# B&R Automation Studio project NAEUL004C00R13L518F00 (part 24)

#### Act_OptP1020Navi.st
```iecst
ACTION Act_OptP1020Navi:

	IF tyP1020McSetNavi.tyNavi.tyBtnMcSet.bRtCompl = TRUE THEN
		tyP1020McSetNavi.tyNavi.tyBtnMcSet.bRtCompl			:= FALSE;
		tyP1020McSetNavi.tyNavi.tyBtnMcSet.bValue			:= FALSE;

		eChgPage	:= UIP1021McSetGen;

	ELSIF tyP1020McSetNavi.tyNavi.tyBtnVCommSet.bRtCompl = TRUE THEN
		tyP1020McSetNavi.tyNavi.tyBtnVCommSet.bRtCompl		:= FALSE;
		tyP1020McSetNavi.tyNavi.tyBtnVCommSet.bValue		:= FALSE;

		eChgPage	:= UIP1022McSetVComm;

	ELSIF tyP1020McSetNavi.tyNavi.tyBtnHCommSet.bRtCompl = TRUE THEN
		tyP1020McSetNavi.tyNavi.tyBtnHCommSet.bRtCompl		:= FALSE;
		tyP1020McSetNavi.tyNavi.tyBtnHCommSet.bValue		:= FALSE;

		eChgPage	:= UIP1023McSetHComm;

	ELSIF tyP1020McSetNavi.tyNavi.tyBtnAntiGapSet.bRtCompl = TRUE THEN
		tyP1020McSetNavi.tyNavi.tyBtnAntiGapSet.bRtCompl	:= FALSE;
		tyP1020McSetNavi.tyNavi.tyBtnAntiGapSet.bValue		:= FALSE;

		eChgPage	:= UIP1024McSetAntiGap;

	ELSIF tyP1020McSetNavi.tyNavi.tyBtnScanSet.bRtCompl = TRUE THEN
		tyP1020McSetNavi.tyNavi.tyBtnScanSet.bRtCompl	:= FALSE;
		tyP1020McSetNavi.tyNavi.tyBtnScanSet.bValue		:= FALSE;

		eChgPage	:= UIP1025McSetScan;

	ELSIF tyP1020McSetNavi.tyNavi.tyBtnOpConSet.bRtCompl = TRUE THEN
		tyP1020McSetNavi.tyNavi.tyBtnOpConSet.bRtCompl	:= FALSE;
		tyP1020McSetNavi.tyNavi.tyBtnOpConSet.bValue		:= FALSE;

		eChgPage	:= UIP1027McSetOpCon;
	END_IF

END_ACTION
```

#### Act_EntP1021Disp.st
```iecst
ACTION Act_EntP1021Disp:

	//Access Address
	IF bTeachTravPosA OR bTeachTravPosB OR bTeachLifterPosA OR bTeachLifterPosB THEN
		p_tyC0004Navi ACCESS ADR(tyP1021McSetGen.tyNaviLyr2);
	ELSIF ((p_tyNtParamCurr.bProjMagConvLane1Prep AND p_tyNtParamCurr.bProjMagConvLane2Prep)
		OR bTeachLifterTopPos OR bTeachLifterTopPos2 OR bTeachLifterBtmPos OR bTeachLifterBtmPos2) OR (p_tyNtParamCurr.tyDISettings.diMagWidthChkSen <>0) THEN
		p_tyC0004Navi ACCESS ADR(tyP1021McSetGen.tyNaviLyr3);
	ELSE
		p_tyC0004Navi ACCESS ADR(tyP1021McSetGen.tyNaviLyr1);
	END_IF

	p_tyC0005Main ACCESS ADR(tyCommon.tyMain);

	p_tyC0006Set ACCESS ADR(tyCommon.tySet);

	p_tyC0007Notif ACCESS ADR(tyCommon.tyNotif);

	p_tyC0008MsgBox ACCESS ADR(tyP1021McSetGen.tyMsgBoxHide);

	p_tyC0009Info ACCESS ADR(tyCommon.tyInfo);

	p_tyP1021McSetGen ACCESS ADR(tyP1021McSetGen.tyGen);
	p_tyP1021McSetNetwork ACCESS ADR(tyP1021McSetGen.tyNetwork);

	//Display
//	tyP1021McSetGen.tyGen.tyLyrGen1.uiRtStat.0	:= bTeachTravPosA OR bTeachTravPosB OR bTeachLifterPosA OR bTeachLifterPosB;
//	tyP1021McSetGen.tyGen.tyLyrGen2.uiRtStat.0	:= NOT(bTeachTravPosA OR bTeachTravPosB OR bTeachLifterPosA OR bTeachLifterPosB);

	//Backup Param
	IF NOT(bTeachTravPosA OR bTeachTravPosB OR bTeachLifterPosA OR bTeachLifterPosB OR
		bTeachLifterTopPos OR bTeachLifterBtmPos OR bTeachLifterTopPos2 OR bTeachLifterBtmPos2) THEN
		tyP1021McSetGen.tyGenBkUp	:= tyP1021McSetGen.tyGen;
	ELSE
		bTeachTravPosA		:= FALSE;
		bTeachTravPosB		:= FALSE;
		bTeachLifterPosA	:= FALSE;
		bTeachLifterPosB	:= FALSE;
		bTeachLifterTopPos	:= FALSE;
		bTeachLifterBtmPos	:= FALSE;
		bTeachLifterTopPos2	:= FALSE;
		bTeachLifterBtmPos2	:= FALSE;
	END_IF
	//Network Configuration Display
	usiNetworkModeOld := DINT_TO_USINT(p_tyMcParamCurr.eNetworkMod);

	fUIInRtStatHide(ADR(tyP1021McSetGen.tyNetwork.tyLyr.uiRtStat));

	IF p_tyDI.bInShutterCloseRS THEN
		tyP1021McSetGen.tyGen.tyBtnInShutterDis.uiMaskRtStat.0 := FALSE;
	ELSE
		tyP1021McSetGen.tyGen.tyBtnInShutterDis.uiMaskRtStat.0 := TRUE;
	END_IF

//	//Penumatic
//	tyP1021McSetGen.tyGen.tyBtnInShutterDis.uiRtStat.0 := TRUE;
	tyP1021McSetGen.tyGen.tyBtnStopperADis.uiRtStat.0 := TRUE;
	tyP1021McSetGen.tyGen.tyBtnStopperBDis.uiRtStat.0 := TRUE;

//	CASE p_tyNtParamCurr.eProjMag OF
//		ULMagDual:
//			tyP1021McSetGen.tyGen.tyStringMcNm.sValue := 'Dual Magazine Line Unloader';
//
//		ULMagTriple:
//			tyP1021McSetGen.tyGen.tyStringMcNm.sValue := 'Triple Magazine Line Unloader';
//
//		ULMagQuadruple:
//			tyP1021McSetGen.tyGen.tyStringMcNm.sValue := 'Quadruple Magazine Line Unloader';
//	END_CASE

	tyP1021McSetGen.tyGen.tyBtnLFBuzMute.uiRtStat.0 := NOT (p_tyMcParamCurr.bLFEn AND p_tyNtParamCurr.bLFPrep AND p_tyNtParamCurr.tyDOSettings.diBuzzer > 0);

	//Siemen Request Hide inlet shutter
	IF p_eNtParamCustomerReq = Siemens THEN
		IF p_tyUsrMgmtCurrAccessRgt.bUsrMgmt THEN
			tyP1021McSetGen.tyGen.tyBtnInShutterDis.uiMaskRtStat := TRUE;
		ELSE
			tyP1021McSetGen.tyGen.tyBtnInShutterDis.uiMaskRtStat := FALSE;
		END_IF
	ELSE
		tyP1021McSetGen.tyGen.tyBtnInShutterDis.uiMaskRtStat := TRUE;
	END_IF
	//Siemen update change for RFID
	tyP1021McSetGen.tyGen.tyBtnMESEn.bValue					:= p_tyMcParamCurr.bMESEn;	//RFID
	tyP1021McSetGen.tyGen.tyBtnHermesSvyEn.bValue					:= p_tyMcParamCurr.bHermesSvyEn;	//RFID

END_ACTION
```

#### Act_ExitP1021.st
```iecst
ACTION Act_ExitP1021:

	IF (tyCommon.tySet.tyBtnSave.uiMaskRtStat.0 = FALSE) OR (bTeachTravPosA OR bTeachTravPosB OR bTeachLifterPosA OR bTeachLifterPosB) THEN
		usiChgPage	:= 1;

	ELSE

		p_tyC0008MsgBox ACCESS ADR(tyP1021McSetGen.tyMsgBoxExitAsk);

		IF tyP1021McSetGen.tyMsgBoxExitAsk.tyBtnYes.bRtCompl = TRUE THEN
			tyP1021McSetGen.tyMsgBoxExitAsk.tyBtnYes.bRtCompl	:= FALSE;
			tyP1021McSetGen.tyMsgBoxExitAsk.tyBtnYes.bValue		:= FALSE;

			p_tyC0008MsgBox ACCESS ADR(tyP1021McSetGen.tyMsgBoxHide);

			//Restore Param
			tyP1021McSetGen.tyGen	:= tyP1021McSetGen.tyGenBkUp;

			fUIInRtStatOff(ADR(tyCommon.tySet.tyBtnSave.uiMaskRtStat));

			bSaveNetworkPriority := FALSE;

			usiChgPage	:= 1;

		ELSIF tyP1021McSetGen.tyMsgBoxExitAsk.tyBtnNo.bRtCompl = TRUE THEN
			tyP1021McSetGen.tyMsgBoxExitAsk.tyBtnNo.bRtCompl	:= FALSE;
			tyP1021McSetGen.tyMsgBoxExitAsk.tyBtnNo.bValue		:= FALSE;

			p_tyC0008MsgBox ACCESS ADR(tyP1021McSetGen.tyMsgBoxHide);

			eChgPage	:= eCurrPage;
			usiChgPage	:= 0;

		END_IF

	END_IF

END_ACTION
```

#### Act_OptP1021Navi.st
```iecst
ACTION Act_OptP1021Navi:

	tyP1021McSetGen.tyNaviLyr1.tyBtnBack.bRtLk	:= tyCommon.tySet.tyBtnSave.bRtCompl;
	tyP1021McSetGen.tyNaviLyr2.tyBtnBack.bRtLk	:= tyCommon.tySet.tyBtnSave.bRtCompl;
	tyP1021McSetGen.tyNaviLyr3.tyBtnBack.bRtLk	:= tyCommon.tySet.tyBtnSave.bRtCompl;

	IF tyP1021McSetGen.tyNaviLyr1.tyBtnBack.bRtCompl = TRUE OR tyP1021McSetGen.tyNaviLyr2.tyBtnBack.bRtCompl = TRUE
		OR tyP1021McSetGen.tyNaviLyr3.tyBtnBack.bRtCompl = TRUE THEN
		tyP1021McSetGen.tyNaviLyr1.tyBtnBack.bRtCompl		:= FALSE;
		tyP1021McSetGen.tyNaviLyr2.tyBtnBack.bRtCompl		:= FALSE;
		tyP1021McSetGen.tyNaviLyr3.tyBtnBack.bRtCompl		:= FALSE;

		eChgPage	:= UIP1020McSetNavi;
	END_IF

	IF (p_tyNtParamCurr.bProjMagConvLane1Prep AND p_tyNtParamCurr.bProjMagConvLane2Prep) OR
		(p_tyNtParamCurr.tyDISettings.diMagWidthChkSen <> 0 OR p_tyNtParamCurr.bProjInletStopperPrep
		OR p_tyNtParamCurr.eCustomerReq = Siemens OR p_tyNtParamCurr.bAutoRcpPrep OR p_tyNtParamCurr.tyDISettings.diScanComplSig <> 0)

		THEN
		p_tyC0004Navi ACCESS ADR (tyP1021McSetGen.tyNaviLyr3);
		IF tyP1021McSetGen.tyNaviLyr3.tyBtnRgt.bRtCompl AND tyP1021McSetGen.tyNaviLyr3.tyBitmapPageDisp.usiValueIdx =3
			OR tyP1021McSetGen.tyNaviLyr3.tyBtnLeft.bRtCompl AND tyP1021McSetGen.tyNaviLyr3.tyBitmapPageDisp.usiValueIdx =5 THEN

			tyP1021McSetGen.tyNaviLyr3.tyBitmapPageDisp.usiValueIdx := 4;
			fUIInRtStatHide(ADR(tyP1021McSetGen.tyGen.tyLyrGen1.uiRtStat));
			fUIInRtStatOff(ADR(tyP1021McSetGen.tyGen.tyLyrGen2.uiRtStat));
			fUIInRtStatHide(ADR(tyP1021McSetGen.tyGen.tyLyrGen3.uiRtStat));
			fUIInRtStatHide(ADR(tyP1021McSetGen.tyGen.tyLyrGen4.uiRtStat));
			tyP1021McSetGen.tyNaviLyr3.tyBtnRgt.bRtCompl := FALSE;
			tyP1021McSetGen.tyNaviLyr3.tyBtnLeft.bRtCompl := FALSE;

		ELSIF tyP1021McSetGen.tyNaviLyr3.tyBtnLeft.bRtCompl AND tyP1021McSetGen.tyNaviLyr3.tyBitmapPageDisp.usiValueIdx =3
			OR tyP1021McSetGen.tyNaviLyr3.tyBtnRgt.bRtCompl AND tyP1021McSetGen.tyNaviLyr3.tyBitmapPageDisp.usiValueIdx =4 THEN

			tyP1021McSetGen.tyNaviLyr3.tyBitmapPageDisp.usiValueIdx := 5;
			fUIInRtStatHide(ADR(tyP1021McSetGen.tyGen.tyLyrGen1.uiRtStat));
			fUIInRtStatHide(ADR(tyP1021McSetGen.tyGen.tyLyrGen2.uiRtStat));
			IF (NOT p_tyNtParamCurr.bProjMagConvLane1Prep AND NOT p_tyNtParamCurr.bProjMagConvLane2Prep)
				AND (p_tyNtParamCurr.tyDISettings.diMagWidthChkSen <> 0 OR p_tyNtParamCurr.bProjInletStopperPrep OR p_tyNtParamCurr.eCustomerReq = Siemens OR  p_tyNtParamCurr.eCustomerReq = We_Fabricate ) THEN
				fUIInRtStatHide(ADR(tyP1021McSetGen.tyGen.tyLyrGen3.uiRtStat));
				fUIInRtStatOff(ADR(tyP1021McSetGen.tyGen.tyLyrGen4.uiRtStat));
			ELSE
				fUIInRtStatOff(ADR(tyP1021McSetGen.tyGen.tyLyrGen3.uiRtStat));
				fUIInRtStatHide(ADR(tyP1021McSetGen.tyGen.tyLyrGen4.uiRtStat));
			END_IF

			tyP1021McSetGen.tyNaviLyr3.tyBtnRgt.bRtCompl := FALSE;
			tyP1021McSetGen.tyNaviLyr3.tyBtnLeft.bRtCompl := FALSE;

		ELSIF (tyP1021McSetGen.tyNaviLyr3.tyBtnLeft.bRtCompl AND tyP1021McSetGen.tyNaviLyr3.tyBitmapPageDisp.usiValueIdx =4)
			OR (tyP1021McSetGen.tyNaviLyr3.tyBtnRgt.bRtCompl AND tyP1021McSetGen.tyNaviLyr3.tyBitmapPageDisp.usiValueIdx =5) THEN

			tyP1021McSetGen.tyNaviLyr3.tyBitmapPageDisp.usiValueIdx := 3;
			fUIInRtStatOff(ADR(tyP1021McSetGen.tyGen.tyLyrGen1.uiRtStat));
			fUIInRtStatHide(ADR(tyP1021McSetGen.tyGen.tyLyrGen2.uiRtStat));
			fUIInRtStatHide(ADR(tyP1021McSetGen.tyGen.tyLyrGen3.uiRtStat));
			fUIInRtStatHide(ADR(tyP1021McSetGen.tyGen.tyLyrGen4.uiRtStat));
			tyP1021McSetGen.tyNaviLyr3.tyBtnRgt.bRtCompl := FALSE;
			tyP1021McSetGen.tyNaviLyr3.tyBtnLeft.bRtCompl := FALSE;
		END_IF

	ELSE

		//Navi From Layer 1 to Layer 2
		IF tyP1021McSetGen.tyNaviLyr1.tyBtnRgt.bRtCompl = TRUE THEN
			p_tyC0004Navi ACCESS ADR (tyP1021McSetGen.tyNaviLyr2);

			fUIInRtStatHide(ADR(tyP1021McSetGen.tyGen.tyLyrGen1.uiRtStat));
			fUIInRtStatOff(ADR(tyP1021McSetGen.tyGen.tyLyrGen2.uiRtStat));

			tyP1021McSetGen.tyNaviLyr1.tyBtnRgt.bRtCompl			:= FALSE;

		ELSIF tyP1021McSetGen.tyNaviLyr1.tyBtnLeft.bRtCompl = TRUE THEN
			p_tyC0004Navi ACCESS ADR (tyP1021McSetGen.tyNaviLyr2);

			fUIInRtStatHide(ADR(tyP1021McSetGen.tyGen.tyLyrGen1.uiRtStat));
			fUIInRtStatOff(ADR(tyP1021McSetGen.tyGen.tyLyrGen2.uiRtStat));

			tyP1021McSetGen.tyNaviLyr1.tyBtnLeft.bRtCompl			:= FALSE;

		//Navi Form Layer 2 to Layer 1
		ELSIF tyP1021McSetGen.tyNaviLyr2.tyBtnRgt.bRtCompl = TRUE THEN
			p_tyC0004Navi ACCESS ADR(tyP1021McSetGen.tyNaviLyr1);

			fUIInRtStatOff(ADR(tyP1021McSetGen.tyGen.tyLyrGen1.uiRtStat));
			fUIInRtStatHide(ADR(tyP1021McSetGen.tyGen.tyLyrGen2.uiRtStat));

			tyP1021McSetGen.tyNaviLyr2.tyBtnRgt.bRtCompl			:= FALSE;

		ELSIF tyP1021McSetGen.tyNaviLyr2.tyBtnLeft.bRtCompl = TRUE THEN
			p_tyC0004Navi ACCESS ADR(tyP1021McSetGen.tyNaviLyr1);

			fUIInRtStatOff(ADR(tyP1021McSetGen.tyGen.tyLyrGen1.uiRtStat));
			fUIInRtStatHide(ADR(tyP1021McSetGen.tyGen.tyLyrGen2.uiRtStat));

			tyP1021McSetGen.tyNaviLyr2.tyBtnLeft.bRtCompl			:= FALSE;

		END_IF
	END_IF

END_ACTION
```

#### Act_OptP1021Save.st
```iecst
ACTION Act_OptP1021Save:
		//Only Applicable when next page appears.

	IF p_tyP1021McSetGen.tyDrpDnPos1.uiRtStat.0 = FALSE
		AND p_tyP1021McSetGen.tyDrpDnPos2.uiRtStat.0 = FALSE
		AND p_tyP1021McSetGen.tyDrpDnPos3.uiRtStat.0 = FALSE THEN

		usiDuplicate := 6;

	ELSIF p_tyP1021McSetGen.tyDrpDnPos1.uiRtStat.0 = FALSE
		AND p_tyP1021McSetGen.tyDrpDnPos2.uiRtStat.0 = FALSE
		AND p_tyP1021McSetGen.tyDrpDnPos3.uiRtStat.0 = TRUE THEN

		usiDuplicate := 3;
	END_IF

	IF tyP1021McSetGen.tyGen.tyStringMcNm.bRtCompl
		OR tyP1021McSetGen.tyGen.tyDrpDnDefaultMcMod.bRtCompl	OR tyP1021McSetGen.tyGen.tyNumSSaverTm.bRtCompl
		OR tyP1021McSetGen.tyGen.tyBtnSSaverEn.bRtCompl			OR tyP1021McSetGen.tyGen.tyNumWidthAtHm.bRtCompl
		OR tyP1021McSetGen.tyGen.tyNumConvInitTm.bRtCompl		OR tyP1021McSetGen.tyGen.tyNumTranInErrDlyTm.bRtCompl
		OR tyP1021McSetGen.tyGen.tyNumMag1ConvRunTm.bRtCompl	OR tyP1021McSetGen.tyGen.tyNumMag2ConvRunTm.bRtCompl
		OR tyP1021McSetGen.tyGen.tyNumMag3ConvRunTm.bRtCompl 	OR tyP1021McSetGen.tyGen.tyNumMaxBffr.bRtCompl
		OR tyP1021McSetGen.tyGen.tyNumTravPosLaneA.bRtCompl		OR tyP1021McSetGen.tyGen.tyNumLiftPosLaneA.bRtCompl
		OR tyP1021McSetGen.tyGen.tyNumTravPosLaneB.bRtCompl		OR tyP1021McSetGen.tyGen.tyNumLiftPosLaneB.bRtCompl
		OR tyP1021McSetGen.tyGen.tyBtnAWDis.bRtCompl			OR tyP1021McSetGen.tyGen.tyBtnMnlAccDat.bRtCompl
		OR tyP1021McSetGen.tyGen.tyBtnAutoStepEn.bRtCompl		OR tyP1021McSetGen.tyGen.tyBtnVSMEMAEn.bRtCompl
		OR tyP1021McSetGen.tyGen.tyBtnHermesRmtEn.bRtCompl		OR tyP1021McSetGen.tyGen.tyBtnGapBetBrdEn.bRtCompl
		OR tyP1021McSetGen.tyGen.tyBtnLongBrdEn.bRtCompl		OR tyP1021McSetGen.tyGen.tyBtnOvenEn.bRtCompl
		OR tyP1021McSetGen.tyGen.tyBtnExtdOvenEn.bRtCompl		OR tyP1021McSetGen.tyGen.tyBtnInShutterDis.bRtCompl
		OR tyP1021McSetGen.tyGen.tyBtnChgParamEn.bRtCompl		OR tyP1021McSetGen.tyGen.tyBtnStopperADis.bRtCompl
		OR tyP1021McSetGen.tyGen.tyBtnStopperBDis.bRtCompl 		OR tyP1021McSetGen.tyGen.tyNumWidthOffset.bRtCompl
		OR tyP1021McSetGen.tyGen.tyBtnAGVComEn.bRtCompl  		OR tyP1021McSetGen.tyGen.tyNumMagAutoDetSenTm.bRtCompl
		OR tyP1021McSetGen.tyGen.tyNumMag1WidthAtHm.bRtCompl	OR tyP1021McSetGen.tyGen.tyNumMag2WidthAtHm.bRtCompl
		OR tyP1021McSetGen.tyGen.tyNumMag3WidthAtHm.bRtCompl	OR tyP1021McSetGen.tyGen.tyBtnMagAWDis.bRtCompl
		OR tyP1021McSetGen.tyGen.tyBtnMagSafetyBarDis.bRtCompl 	OR tyP1021McSetGen.tyGen.tyBtnAutoLogoutEn.bRtCompl
		OR tyP1021McSetGen.tyGen.tyNumAutoLogoutTm.bRtCompl		OR tyP1021McSetGen.tyGen.tyBtnLFBuzMute.bRtCompl
		OR tyP1021McSetGen.tyGen.tyDrpDnAGVComProtocol.bRtCompl OR tyP1021McSetGen.tyGen.tyDrpDnMagExchangeMode.bRtCompl
		OR tyP1021McSetGen.tyGen.tyBtnAGVSizeDisabled.bRtCompl
		OR tyP1021McSetGen.tyGen.tyNumAWPusherAtHm.bRtCompl		OR tyP1021McSetGen.tyGen.tyBtnAWPusherDis.bRtCompl
		OR tyP1021McSetGen.tyGen.tyNumTravFixtoFixPosInlet.bRtCompl
		OR tyP1021McSetGen.tyGen.tyBtnDisableFMWarning.bRtCompl
		OR tyP1021McSetGen.tyGen.tyNumInMagConvInitTm.bRtCompl OR tyP1021McSetGen.tyGen.tyNumOutMagConvInitTm.bRtCompl
		OR tyP1021McSetGen.tyGen.tyNumLifterTopPos.bRtCompl OR tyP1021McSetGen.tyGen.tyNumLifterBtmPos.bRtCompl
		OR tyP1021McSetGen.tyGen.tyNumLifterMagConvInitTm.bRtCompl
		OR tyP1021McSetGen.tyGen.tyNumInMagConv2InitTm.bRtCompl OR tyP1021McSetGen.tyGen.tyNumOutMagConv2InitTm.bRtCompl
		OR tyP1021McSetGen.tyGen.tyNumLifterTopPos2.bRtCompl OR tyP1021McSetGen.tyGen.tyNumLifterBtmPos2.bRtCompl
		OR tyP1021McSetGen.tyGen.tyNumLifterMagConv2InitTm.bRtCompl OR tyP1021McSetGen.tyGen.tyNumTCPSvrPort.bRtCompl
		OR tyP1021McSetGen.tyGen.tyBtnMagWidthChkDis.bRtCompl OR tyP1021McSetGen.tyGen.tyNumMag1WidthChkDetDist.bRtCompl
		OR tyP1021McSetGen.tyGen.tyNumMag2WidthChkDetDist.bRtCompl OR tyP1021McSetGen.tyGen.tyNumMag3WidthChkDetDist.bRtCompl
		OR tyP1021McSetGen.tyGen.tyBtnHermesSvyEn.bRtCompl OR tyP1021McSetGen.tyGen.tyBtnInletStopperDis.bRtCompl
		OR tyP1021McSetGen.tyGen.tyNumMESResponseTO.bRtCompl OR tyP1021McSetGen.tyGen.tyBtnMESEn.bRtCompl
		OR tyP1021McSetGen.tyGen.tyBtnSwitchingProductType.bRtCompl OR tyP1021McSetGen.tyGen.tyNumInStprDelayTm.bRtCompl
		OR tyP1021McSetGen.tyGen.tyBtnBatchIDChgOverCmp.bRtCompl OR tyP1021McSetGen.tyGen.tyBtnIgnoreTopClearance.bRtCompl
		OR tyP1021McSetGen.tyGen.tyBtnIgnoreBottomClearance.bRtCompl OR tyP1021McSetGen.tyGen.tyBtnIgnoreThickness.bRtCompl
		OR tyP1021McSetGen.tyGen.tyBtnDMCScannerEn.bRtCompl OR tyP1021McSetGen.tyGen.tyNumDMCScanWriteTO.bRtCompl
		OR tyP1021McSetGen.tyGen.tyDrpDnPos1.bRtCompl OR tyP1021McSetGen.tyGen.tyDrpDnPos2.bRtCompl
		OR tyP1021McSetGen.tyGen.tyDrpDnPos3.bRtCompl OR tyP1021McSetGen.tyGen.tyStringDefaultGWIP.bRtCompl
		THEN

		fUIInRtStatHide(ADR(tyCommon.tySet.tyBtnSave.uiMaskRtStat));

		tyP1021McSetGen.tyGen.tyStringMcNm.bRtCompl			:= FALSE;
		tyP1021McSetGen.tyGen.tyDrpDnDefaultMcMod.bRtCompl	:= FALSE;
		tyP1021McSetGen.tyGen.tyNumSSaverTm.bRtCompl		:= FALSE;
		tyP1021McSetGen.tyGen.tyBtnSSaverEn.bRtCompl		:= FALSE;
		tyP1021McSetGen.tyGen.tyNumWidthAtHm.bRtCompl		:= FALSE;
		tyP1021McSetGen.tyGen.tyNumConvInitTm.bRtCompl		:= FALSE;
		tyP1021McSetGen.tyGen.tyNumTranInErrDlyTm.bRtCompl	:= FALSE;
		tyP1021McSetGen.tyGen.tyNumMag1ConvRunTm.bRtCompl	:= FALSE;
		tyP1021McSetGen.tyGen.tyNumMag2ConvRunTm.bRtCompl	:= FALSE;
		tyP1021McSetGen.tyGen.tyNumMag3ConvRunTm.bRtCompl 	:= FALSE;
		tyP1021McSetGen.tyGen.tyNumMaxBffr.bRtCompl			:= FALSE;
		tyP1021McSetGen.tyGen.tyBtnAGVComEn.bRtCompl		:= FALSE;
		tyP1021McSetGen.tyGen.tyNumMag1WidthAtHm.bRtCompl	:= FALSE;
		tyP1021McSetGen.tyGen.tyNumMag2WidthAtHm.bRtCompl	:= FALSE;
		tyP1021McSetGen.tyGen.tyNumMag3WidthAtHm.bRtCompl	:= FALSE;

		tyP1021McSetGen.tyGen.tyNumTravPosLaneA.bRtCompl	:= FALSE;
		tyP1021McSetGen.tyGen.tyNumLiftPosLaneA.bRtCompl	:= FALSE;
		tyP1021McSetGen.tyGen.tyNumTravPosLaneB.bRtCompl	:= FALSE;
		tyP1021McSetGen.tyGen.tyNumLiftPosLaneB.bRtCompl	:= FALSE;
		tyP1021McSetGen.tyGen.tyBtnAWDis.bRtCompl			:= FALSE;
		tyP1021McSetGen.tyGen.tyBtnMnlAccDat.bRtCompl		:= FALSE;
		tyP1021McSetGen.tyGen.tyBtnAutoStepEn.bRtCompl		:= FALSE;
		tyP1021McSetGen.tyGen.tyBtnVSMEMAEn.bRtCompl		:= FALSE;
		tyP1021McSetGen.tyGen.tyBtnHermesRmtEn.bRtCompl		:= FALSE;
		tyP1021McSetGen.tyGen.tyBtnGapBetBrdEn.bRtCompl		:= FALSE;
		tyP1021McSetGen.tyGen.tyBtnLongBrdEn.bRtCompl		:= FALSE;
		tyP1021McSetGen.tyGen.tyBtnOvenEn.bRtCompl			:= FALSE;
		tyP1021McSetGen.tyGen.tyBtnExtdOvenEn.bRtCompl		:= FALSE;
		tyP1021McSetGen.tyGen.tyBtnInShutterDis.bRtCompl	:= FALSE;
		tyP1021McSetGen.tyGen.tyBtnChgParamEn.bRtCompl		:= FALSE;
		tyP1021McSetGen.tyGen.tyBtnStopperADis.bRtCompl		:= FALSE;
		tyP1021McSetGen.tyGen.tyBtnStopperBDis.bRtCompl		:= FALSE;
		tyP1021McSetGen.tyGen.tyNumWidthOffset.bRtCompl		:= FALSE;
		tyP1021McSetGen.tyGen.tyNumMagAutoDetSenTm.bRtCompl	 := FALSE;
		tyP1021McSetGen.tyGen.tyBtnMagAWDis.bRtCompl		:= FALSE;
		tyP1021McSetGen.tyGen.tyBtnMagSafetyBarDis.bRtCompl	:= FALSE;
		tyP1021McSetGen.tyGen.tyBtnAutoLogoutEn.bRtCompl	:= FALSE;
		tyP1021McSetGen.tyGen.tyNumAutoLogoutTm.bRtCompl	:= FALSE;
		tyP1021McSetGen.tyGen.tyBtnLFBuzMute.bRtCompl		:= FALSE;
		tyP1021McSetGen.tyGen.tyDrpDnAGVComProtocol.bRtCompl:= FALSE;
		tyP1021McSetGen.tyGen.tyDrpDnMagExchangeMode.bRtCompl := FALSE;
		tyP1021McSetGen.tyGen.tyBtnAGVSizeDisabled.bRtCompl := FALSE;
		tyP1021McSetGen.tyGen.tyBtnMagWidthChkDis.bRtCompl	:= FALSE;
		tyP1021McSetGen.tyGen.tyBtnDMCScannerEn.bRtCompl 		:= FALSE;
		tyP1021McSetGen.tyGen.tyNumDMCScanWriteTO.bRtCompl	:= FALSE;

		tyP1021McSetGen.tyGen.tyNumAWPusherAtHm.bRtCompl	:= FALSE;
		tyP1021McSetGen.tyGen.tyBtnAWPusherDis.bRtCompl		:= FALSE;
		tyP1021McSetGen.tyGen.tyNumTravFixtoFixPosInlet.bRtCompl:= FALSE;
		tyP1021McSetGen.tyGen.tyBtnDisableFMWarning.bRtCompl:= FALSE;
		tyP1021McSetGen.tyGen.tyNumInMagConvInitTm.bRtCompl := FALSE;
		tyP1021McSetGen.tyGen.tyNumOutMagConvInitTm.bRtCompl := FALSE;
		tyP1021McSetGen.tyGen.tyNumLifterTopPos.bRtCompl := FALSE;
		tyP1021McSetGen.tyGen.tyNumLifterBtmPos.bRtCompl := FALSE;
		tyP1021McSetGen.tyGen.tyNumLifterMagConvInitTm.bRtCompl := FALSE;
		tyP1021McSetGen.tyGen.tyNumInMagConv2InitTm.bRtCompl := FALSE;
		tyP1021McSetGen.tyGen.tyNumOutMagConv2InitTm.bRtCompl := FALSE;
		tyP1021McSetGen.tyGen.tyNumLifterTopPos2.bRtCompl := FALSE;
		tyP1021McSetGen.tyGen.tyNumLifterBtmPos2.bRtCompl := FALSE;
		tyP1021McSetGen.tyGen.tyNumLifterMagConv2InitTm.bRtCompl := FALSE;
		tyP1021McSetGen.tyGen.tyNumTCPSvrPort.bRtCompl	:= FALSE;
		tyP1021McSetGen.tyGen.tyNumMag1WidthChkDetDist.bRtCompl	:= FALSE;
		tyP1021McSetGen.tyGen.tyNumMag2WidthChkDetDist.bRtCompl	:= FALSE;
		tyP1021McSetGen.tyGen.tyNumMag3WidthChkDetDist.bRtCompl	:= FALSE;

		tyP1021McSetGen.tyGen.tyBtnHermesSvyEn.bRtCompl		:= FALSE;
		tyP1021McSetGen.tyGen.tyBtnInletStopperDis.bRtCompl	:= FALSE;
		tyP1021McSetGen.tyGen.tyNumMESResponseTO.bRtCompl	:= FALSE;
		tyP1021McSetGen.tyGen.tyBtnMESEn.bRtCompl		:= FALSE;
		tyP1021McSetGen.tyGen.tyBtnSwitchingProductType.bRtCompl := FALSE;
		tyP1021McSetGen.tyGen.tyBtnBatchIDChgOverCmp.bRtCompl := FALSE;
		tyP1021McSetGen.tyGen.tyBtnIgnoreTopClearance.bRtCompl := FALSE;
		tyP1021McSetGen.tyGen.tyBtnIgnoreBottomClearance.bRtCompl := FALSE;
		tyP1021McSetGen.tyGen.tyBtnIgnoreThickness.bRtCompl := FALSE;
		tyP1021McSetGen.tyGen.tyStringDefaultGWIP.bRtCompl := FALSE;
		//Added Main Menu
		tyP1021McSetGen.tyGen.tyDrpDnPos1.bRtCompl				:= FALSE;
		tyP1021McSetGen.tyGen.tyDrpDnPos2.bRtCompl				:= FALSE;
		tyP1021McSetGen.tyGen.tyDrpDnPos3.bRtCompl				:= FALSE;
	END_IF

	IF tyCommon.tySet.tyBtnSave.bRtCompl = TRUE AND bSaveNetworkPriority=FALSE THEN
		IF usiGenSaveStep = 0 THEN
//			IF (p_tyP1021McSetGen.tyDrpDnPos1.usiValueIdx + p_tyP1021McSetGen.tyDrpDnPos2.usiValueIdx + p_tyP1021McSetGen.tyDrpDnPos3.usiValueIdx <> usiDuplicate)
//				AND p_tyNtParamCurr.tyUIBtnPosLmt.diMax <> 1 THEN
//				usiGenSaveStep := 99;
//			ELSE
				usiGenSaveStep := 1;
//			END_IF
		ELSIF usiGenSaveStep = 1 THEN

			tyMcParamWr.sMcNm					:=	tyP1021McSetGen.tyGen.tyStringMcNm.sValue;
			tyMcParamWr.usiDefaultMcMod			:=	tyP1021McSetGen.tyGen.tyDrpDnDefaultMcMod.usiValueIdx;
			tyMcParamWr.uiSSaverTmInSec			:= 	DINT_TO_UINT(tyP1021McSetGen.tyGen.tyNumSSaverTm.diValue);
			tyMcParamWr.bSSaverEn				:=	tyP1021McSetGen.tyGen.tyBtnSSaverEn.bValue;
			tyMcParamWr.diWidthAtHmPosInUM		:=	tyP1021McSetGen.tyGen.tyNumWidthAtHm.diValue;
			tyMcParamWr.diConvInitTmInMS		:=	tyP1021McSetGen.tyGen.tyNumConvInitTm.diValue;
			tyMcParamWr.diTranInErrDlyTmInMS	:=	tyP1021McSetGen.tyGen.tyNumTranInErrDlyTm.diValue;
			tyMcParamWr.diMag1ConvRunTmOutInMS	:=	tyP1021McSetGen.tyGen.tyNumMag1ConvRunTm.diValue;
			tyMcParamWr.diMag2ConvRunTmOutInMS	:=	tyP1021McSetGen.tyGen.tyNumMag2ConvRunTm.diValue;
			tyMcParamWr.diMag3ConvRunTmOutInMS	:=	tyP1021McSetGen.tyGen.tyNumMag3ConvRunTm.diValue;
			tyMcParamWr.diOvenMaxBffr			:=  tyP1021McSetGen.tyGen.tyNumMaxBffr.diValue;
			tyMcParamWr.diMagAutoDetectSenTmInMS:=  tyP1021McSetGen.tyGen.tyNumMagAutoDetSenTm.diValue;
			tyMcParamWr.diMag1WidthAtHmPosInUM	:=	tyP1021McSetGen.tyGen.tyNumMag1WidthAtHm.diValue;
			tyMcParamWr.diMag2WidthAtHmPosInUM	:=	tyP1021McSetGen.tyGen.tyNumMag2WidthAtHm.diValue;
			tyMcParamWr.diMag3WidthAtHmPosInUM	:=	tyP1021McSetGen.tyGen.tyNumMag3WidthAtHm.diValue;

			tyMcParamWr.diTravPosA				:=	tyP1021McSetGen.tyGen.tyNumTravPosLaneA.diValue;
			tyMcParamWr.diLifterPosA			:=	tyP1021McSetGen.tyGen.tyNumLiftPosLaneA.diValue;
			tyMcParamWr.diTravPosB				:=	tyP1021McSetGen.tyGen.tyNumTravPosLaneB.diValue;
			tyMcParamWr.diLifterPosB			:=	tyP1021McSetGen.tyGen.tyNumLiftPosLaneB.diValue;
			tyMcParamWr.bAWDis					:=	tyP1021McSetGen.tyGen.tyBtnAWDis.bValue;
			tyMcParamWr.bMnlAccDat				:=	tyP1021McSetGen.tyGen.tyBtnMnlAccDat.bValue;
			tyMcParamWr.bAutoStepEn				:=	tyP1021McSetGen.tyGen.tyBtnAutoStepEn.bValue;
			tyMcParamWr.bVSMEMAEn				:=	tyP1021McSetGen.tyGen.tyBtnVSMEMAEn.bValue;
			tyMcParamWr.bHermesRmtEn			:=	tyP1021McSetGen.tyGen.tyBtnHermesRmtEn.bValue;
			tyMcParamWr.bHermesSvyEn			:= tyP1021McSetGen.tyGen.tyBtnHermesSvyEn.bValue;//new for Hermes 1.3
			tyMcParamWr.bGapBwtnBrdEn			:=  tyP1021McSetGen.tyGen.tyBtnGapBetBrdEn.bValue;
			tyMcParamWr.bLongBrdEn				:=  tyP1021McSetGen.tyGen.tyBtnLongBrdEn.bValue;
			tyMcParamWr.bOvenEn					:=  tyP1021McSetGen.tyGen.tyBtnOvenEn.bValue;
			tyMcParamWr.bExtdOvenEn				:=  tyP1021McSetGen.tyGen.tyBtnExtdOvenEn.bValue;
			tyMcParamWr.bInShutterDis			:=  tyP1021McSetGen.tyGen.tyBtnInShutterDis.bValue;
			tyMcParamWr.bChgParamEn				:=  tyP1021McSetGen.tyGen.tyBtnChgParamEn.bValue;
			tyMcParamWr.bStopperADis			:=  tyP1021McSetGen.tyGen.tyBtnStopperADis.bValue;
			tyMcParamWr.bStopperBDis			:=  tyP1021McSetGen.tyGen.tyBtnStopperBDis.bValue;
			tyMcParamWr.diWidthOffsetInUM		:= 	tyP1021McSetGen.tyGen.tyNumWidthOffset.diValue;
			tyMcParamWr.bAGVComEn				:=  tyP1021McSetGen.tyGen.tyBtnAGVComEn.bValue;
			tyMcParamWr.eNetworkMod				:= 	USINT_TO_DINT(tyP1021McSetGen.tyGen.tyDrpDnNetworkMod.usiValueIdx);
			tyMcParamWr.bMagAWDis				:=  tyP1021McSetGen.tyGen.tyBtnMagAWDis.bValue;
			tyMcParamWr.bMagSafetyBarDis		:=  tyP1021McSetGen.tyGen.tyBtnMagSafetyBarDis.bValue;
			tyMcParamWr.bAutoLogoutEn			:=	tyP1021McSetGen.tyGen.tyBtnAutoLogoutEn.bValue;
			tyMcParamWr.diAutoLogoutTmInSec		:=	tyP1021McSetGen.tyGen.tyNumAutoLogoutTm.diValue;
			tyMcParamWr.bLFBuzMute				:=  tyP1021McSetGen.tyGen.tyBtnLFBuzMute.bValue;
			tyMcParamWr.eAGVComProtocol			:=  tyP1021McSetGen.tyGen.tyDrpDnAGVComProtocol.usiValueIdx;
			tyMcParamWr.eMagExMode				:=  tyP1021McSetGen.tyGen.tyDrpDnMagExchangeMode.usiValueIdx;
			tyMcParamWr.bAIVSizeDisabled		:=  tyP1021McSetGen.tyGen.tyBtnAGVSizeDisabled.bValue;
			tyMcParamWr.bMagWidthChkDis			:=  tyP1021McSetGen.tyGen.tyBtnMagWidthChkDis.bValue;
			tyMcParamWr.bDMCScannerEn			:=  tyP1021McSetGen.tyGen.tyBtnDMCScannerEn.bValue;
			tyMcParamWr.diDMCScanTOErrInMs		:=  tyP1021McSetGen.tyGen.tyNumDMCScanWriteTO.diValue;

			tyMcParamWr.diAWPusherAtHmPosInUM	:=	tyP1021McSetGen.tyGen.tyNumAWPusherAtHm.diValue;
			tyMcParamWr.bAWPusherDis			:=	tyP1021McSetGen.tyGen.tyBtnAWPusherDis.bValue;

			tyMcParamWr.diTravInletFixtoFixPos	:=  tyP1021McSetGen.tyGen.tyNumTravFixtoFixPosInlet.diValue;
			tyMcParamWr.bDisableFMWarning		:= 	tyP1021McSetGen.tyGen.tyBtnDisableFMWarning.bValue;

			tyMcParamWr.diInMagConvRunTmOutInMS			:= 	tyP1021McSetGen.tyGen.tyNumInMagConvInitTm.diValue;
			tyMcParamWr.diOutMagConvRunTmOutInMS		:= 	tyP1021McSetGen.tyGen.tyNumOutMagConvInitTm.diValue;
			tyMcParamWr.diLifterMagConvRunTmOutInMS		:=	tyP1021McSetGen.tyGen.tyNumLifterMagConvInitTm.diValue;
			tyMcParamWr.diLifterTopPos					:=	tyP1021McSetGen.tyGen.tyNumLifterTopPos.diValue;
			tyMcParamWr.diLifterBtmPos					:=	tyP1021McSetGen.tyGen.tyNumLifterBtmPos.diValue;

			tyMcParamWr.diInMagConv2RunTmOutInMS		:= 	tyP1021McSetGen.tyGen.tyNumInMagConv2InitTm.diValue;
			tyMcParamWr.diOutMagConv2RunTmOutInMS		:= 	tyP1021McSetGen.tyGen.tyNumOutMagConv2InitTm.diValue;
			tyMcParamWr.diLifterMagConv2RunTmOutInMS	:=	tyP1021McSetGen.tyGen.tyNumLifterMagConv2InitTm.diValue;
			tyMcParamWr.diLifterTopPos2					:=	tyP1021McSetGen.tyGen.tyNumLifterTopPos2.diValue;
			tyMcParamWr.diLifterBtmPos2					:=	tyP1021McSetGen.tyGen.tyNumLifterBtmPos2.diValue;
			tyMcParamWr.diTCPSvrPort					:=	tyP1021McSetGen.tyGen.tyNumTCPSvrPort.diValue;

			tyMcParamWr.diMag1WidthChkDetDist			:=	tyP1021McSetGen.tyGen.tyNumMag1WidthChkDetDist.diValue;
			tyMcParamWr.diMag2WidthChkDetDist			:=	tyP1021McSetGen.tyGen.tyNumMag2WidthChkDetDist.diValue;
			tyMcParamWr.diMag3WidthChkDetDist			:=	tyP1021McSetGen.tyGen.tyNumMag3WidthChkDetDist.diValue;

			tyMcParamWr.diMag1WidthChkDetDist			:=	tyP1021McSetGen.tyGen.tyNumMag1WidthChkDetDist.diValue;
			tyMcParamWr.diMag2WidthChkDetDist			:=	tyP1021McSetGen.tyGen.tyNumMag2WidthChkDetDist.diValue;
			tyMcParamWr.diMag3WidthChkDetDist			:=	tyP1021McSetGen.tyGen.tyNumMag3WidthChkDetDist.diValue;

			tyMcParamWr.bInStopperDis					:=	tyP1021McSetGen.tyGen.tyBtnInletStopperDis.bValue;
			tyMcParamWr.diInletStopperExtDelayTmInMS	:= 	tyP1021McSetGen.tyGen.tyNumInStprDelayTm.diValue;
			tyMcParamWr.diMESResponseTOTmInMS			:= 	tyP1021McSetGen.tyGen.tyNumMESResponseTO.diValue;
			tyMcParamWr.bMESEn							:=	tyP1021McSetGen.tyGen.tyBtnMESEn.bValue;
			tyMcParamWr.bSwitchingProdType				:=	tyP1021McSetGen.tyGen.tyBtnSwitchingProductType.bValue; //for AutoRcp and Traverser
			tyMcParamWr.bBatchIDChgOverCmp				:= 	tyP1021McSetGen.tyGen.tyBtnBatchIDChgOverCmp.bRtCompl;
			tyMcParamWr.bIgnoreTopClearance				:= 	tyP1021McSetGen.tyGen.tyBtnIgnoreTopClearance.bRtCompl;
			tyMcParamWr.bIgnoreBtmClearance				:= 	tyP1021McSetGen.tyGen.tyBtnIgnoreBottomClearance.bRtCompl;
			tyMcParamWr.bIgnoreThickness				:= 	tyP1021McSetGen.tyGen.tyBtnIgnoreThickness.bRtCompl;

			IF fIPValid(tyP1021McSetGen.tyGen.tyStringDefaultGWIP.sValue,ADR(a_iIPPart1)) THEN
				tyMcParamWr.sDefaultGateWay := tyP1021McSetGen.tyGen.tyStringDefaultGWIP.sValue;
			ELSE
				tyP1021McSetGen.tyGen.tyStringDefaultGWIP.sValue := '0.0.0.0';
				tyMcParamWr.sDefaultGateWay := '0.0.0.0';
			END_IF

			IF tyP1021McSetGen.tyGen.tyDrpDnNetworkMod.usiValueIdx =DINT_TO_USINT(SetIPManually) THEN
				tyMcParamWr.sIPAddr				:= tyP1021McSetGen.tyGen.tyStringIPAddr.sValue;
				tyMcParamWr.sSubnetMask			:= tyP1021McSetGen.tyGen.tyStringSubnetMask.sValue;
				//ADD
				tyMcParamWr.sHMIIPAddr			:= tyP1021McSetGen.tyGen.tyStringHMIIPAddr.sValue;
			END_IF

			eMcParamAct	:= McParamActWrite;

			IF p_eMcParamStat = McParamActWrite AND p_eMcParamStatus = Done THEN
				eMcParamAct	:= McParamActIdle;
				eHWInfoAct := HWInfoActSetDefaultGateway;

				usiNetworkModeOld := tyP1021McSetGen.tyGen.tyDrpDnNetworkMod.usiValueIdx;
				//Screen Saver Time
				tyProperty.tyVisu.uiSSaverTm	:= p_tyMcParamCurr.uiSSaverTmInSec;

				//Backup Param
				tyP1021McSetGen.tyGenBkUp	:= tyP1021McSetGen.tyGen;

				tyCommon.tySet.tyBtnSave.bRtCompl 	:= FALSE;
				fUIInRtStatOff(ADR(tyCommon.tySet.tyBtnSave.uiMaskRtStat));
				usiGenSaveStep := 0;
			ELSIF p_eMcParamStatus = Error THEN
				p_tyC0008MsgBox ACCESS ADR(tyP1021McSetGen.tyMsgBoxSaveErr);

				IF tyP1021McSetGen.tyMsgBoxSaveErr.tyBtnNo.bRtCompl = TRUE THEN
					tyP1021McSetGen.tyMsgBoxSaveErr.tyBtnNo.bRtCompl	:= FALSE;
					tyP1021McSetGen.tyMsgBoxSaveErr.tyBtnNo.bValue		:= FALSE;

					p_tyC0008MsgBox ACCESS ADR(tyP1021McSetGen.tyMsgBoxHide);

					//Restore Param
					tyP1021McSetGen.tyGen	:= tyP1021McSetGen.tyGenBkUp;
					tyMcParamWr				:= p_tyMcParamCurr;

					tyCommon.tySet.tyBtnSave.bRtCompl 	:= FALSE;
					fUIInRtStatOff(ADR(tyCommon.tySet.tyBtnSave.uiMaskRtStat));
					usiGenSaveStep := 0;
				END_IF
			END_IF
		ELSIF usiGenSaveStep = 99 THEN
			p_tyC0008MsgBox ACCESS ADR(tyP1021McSetGen.tyMsgBoxBtnPosDuplicate);

			IF tyP1021McSetGen.tyMsgBoxBtnPosDuplicate.tyBtnNo.bRtCompl = TRUE THEN
				tyP1021McSetGen.tyMsgBoxBtnPosDuplicate.tyBtnNo.bRtCompl := FALSE;
				tyP1021McSetGen.tyMsgBoxBtnPosDuplicate.tyBtnNo.bValue   := FALSE;

				p_tyC0008MsgBox ACCESS ADR(tyP1021McSetGen.tyMsgBoxHide);

				tyCommon.tySet.tyBtnSave.bRtCompl := FALSE;
				usiGenSaveStep := 0;
			END_IF

		END_IF

	ELSIF bUpdateP1021Network THEN
		tyMcParamWr.sIPAddr					:= tyP1021McSetGen.tyGen.tyStringIPAddr.sValue;
		tyMcParamWr.sSubnetMask				:= tyP1021McSetGen.tyGen.tyStringSubnetMask.sValue;
		//ADD
		tyMcParamWr.sHMIIPAddr				:= tyP1021McSetGen.tyGen.tyStringHMIIPAddr.sValue;

		eMcParamAct	:= McParamActWrite;

		IF p_eMcParamStat = McParamActWrite AND p_eMcParamStatus = Done THEN
			eMcParamAct		:= McParamActIdle;
			//ADD
			IF bUpdtHMIIPAddr = FALSE THEN
				eMcParamAct		:= McParamActIdle;
			END_IF

			IF bUpdateP1021Network THEN
				bUpdateP1021Network :=FALSE;
			END_IF

			//Update Restore Param
			tyP1021McSetGen.tyGenBkUp.tyStringIPAddr.sValue	 	:= tyP1021McSetGen.tyGen.tyStringIPAddr.sValue;
			tyP1021McSetGen.tyGenBkUp.tyStringSubnetMask.sValue	:= tyP1021McSetGen.tyGen.tyStringSubnetMask.sValue;
			sDefaultGWBlkUp := '0.0.0.0';
			//ADD
			tyP1021McSetGen.tyGenBkUp.tyStringHMIIPAddr.sValue	:= tyP1021McSetGen.tyGen.tyStringHMIIPAddr.sValue;

		ELSIF p_eMcParamStatus = Error THEN
			p_tyC0008MsgBox ACCESS ADR(tyP1021McSetGen.tyMsgBoxSaveErr);

			IF tyP1021McSetGen.tyMsgBoxSaveErr.tyBtnNo.bRtCompl = TRUE THEN
				tyP1021McSetGen.tyMsgBoxSaveErr.tyBtnNo.bRtCompl 			:= FALSE;
				tyP1021McSetGen.tyMsgBoxSaveErr.tyBtnNo.bValue				:= FALSE;

				p_tyC0008MsgBox ACCESS ADR(tyP1021McSetGen.tyMsgBoxHide);

				// Restore Param
				tyP1021McSetGen.tyGenBkUp.tyStringIPAddr.sValue	 	:= tyP1021McSetGen.tyGen.tyStringIPAddr.sValue;
				tyP1021McSetGen.tyGenBkUp.tyStringSubnetMask.sValue	:= tyP1021McSetGen.tyGen.tyStringSubnetMask.sValue;
				//ADD
				tyP1021McSetGen.tyGenBkUp.tyStringHMIIPAddr.sValue	:= tyP1021McSetGen.tyGen.tyStringHMIIPAddr.sValue;
				tyMcParamWr				:= p_tyMcParamCurr;

				bUpdateP1021Network :=FALSE;

			END_IF
		END_IF
	END_IF

	IF p_eHWInfoStat = HWInfoActSetDefaultGateway AND p_eHWInfoStatus = Done THEN
		eHWInfoAct	:= HWInfoActIdle;
		sDefaultGWBlkUp := tyP1021McSetGen.tyGen.tyStringDefaultGWIP.sValue;
	ELSIF p_eHWInfoStat = HWInfoActSetDefaultGateway AND p_eHWInfoStatus = Error AND NOT(tyP1021McSetGen.tyMsgBoxSetDefaultGWErr.tyBtnNo.bValue) THEN
		p_tyC0008MsgBox ACCESS ADR(tyP1021McSetGen.tyMsgBoxSetDefaultGWErr);
		tyP1021McSetGen.tyGen.tyStringDefaultGWIP.sValue := sDefaultGWBlkUp;
	ELSIF p_eHWInfoStatus = Idle THEN
		tyP1021McSetGen.tyMsgBoxSetDefaultGWErr.tyBtnNo.bValue := FALSE;
	END_IF

	IF tyP1021McSetGen.tyMsgBoxSetDefaultGWErr.tyBtnNo.bRtCompl = TRUE THEN
		tyP1021McSetGen.tyMsgBoxSetDefaultGWErr.tyBtnNo.bRtCompl	:= FALSE;
		tyCommon.tyMain.tyBtnReset.bRtCompl := TRUE;
		p_tyC0008MsgBox ACCESS ADR(tyP1021McSetGen.tyMsgBoxHide);
		tyCommon.tySet.tyBtnSave.bRtCompl := TRUE;
	END_IF

END_ACTION
```

#### Act_OptP1021Teach.st
```iecst
ACTION Act_OptP1021Teach:

	IF tyP1021McSetGen.tyGen.tyBtnTravPosATeach.bRtCompl = TRUE THEN
		tyP1021McSetGen.tyGen.tyBtnTravPosATeach.bRtCompl	:= FALSE;
		tyP1021McSetGen.tyGen.tyBtnTravPosATeach.bValue		:= FALSE;

		bTeachTravPosA  	:= TRUE;
		eChgPage			:= UIP1026McSetTeach;

	ELSIF tyP1021McSetGen.tyGen.tyBtnTravPosBTeach.bRtCompl = TRUE THEN
		tyP1021McSetGen.tyGen.tyBtnTravPosBTeach.bRtCompl	:= FALSE;
		tyP1021McSetGen.tyGen.tyBtnTravPosBTeach.bValue		:= FALSE;

		bTeachTravPosB		:= TRUE;
		eChgPage			:= UIP1026McSetTeach;

	ELSIF tyP1021McSetGen.tyGen.tyBtnLiftPosATeach.bRtCompl = TRUE THEN
		tyP1021McSetGen.tyGen.tyBtnLiftPosATeach.bRtCompl	:= FALSE;
		tyP1021McSetGen.tyGen.tyBtnLiftPosATeach.bValue		:= FALSE;

		bTeachLifterPosA	:= TRUE;
		eChgPage			:= UIP1026McSetTeach;

	ELSIF tyP1021McSetGen.tyGen.tyBtnLiftPosBTeach.bRtCompl = TRUE THEN
		tyP1021McSetGen.tyGen.tyBtnLiftPosBTeach.bRtCompl	:= FALSE;
		tyP1021McSetGen.tyGen.tyBtnLiftPosBTeach.bValue		:= FALSE;

		bTeachLifterPosB	:= TRUE;
		eChgPage			:= UIP1026McSetTeach;

	ELSIF tyP1021McSetGen.tyGen.tyBtnTeachTopPos.bRtCompl = TRUE THEN //LifterConv
		tyP1021McSetGen.tyGen.tyBtnTeachTopPos.bRtCompl		:= FALSE;
		tyP1021McSetGen.tyGen.tyBtnTeachTopPos.bValue		:= FALSE;

		bTeachLifterTopPos	:= TRUE;
		eChgPage			:= UIP1026McSetTeach;
	ELSIF tyP1021McSetGen.tyGen.tyBtnTeachBtmPos.bRtCompl = TRUE THEN
		tyP1021McSetGen.tyGen.tyBtnTeachBtmPos.bRtCompl		:= FALSE;
		tyP1021McSetGen.tyGen.tyBtnTeachBtmPos.bValue		:= FALSE;

		bTeachLifterBtmPos	:= TRUE;
		eChgPage			:= UIP1026McSetTeach;

	ELSIF tyP1021McSetGen.tyGen.tyBtnTeachTopPos2.bRtCompl = TRUE THEN
		tyP1021McSetGen.tyGen.tyBtnTeachTopPos2.bRtCompl	:= FALSE;
		tyP1021McSetGen.tyGen.tyBtnTeachTopPos2.bValue		:= FALSE;

		bTeachLifterTopPos2	:= TRUE;
		eChgPage			:= UIP1026McSetTeach;
	ELSIF tyP1021McSetGen.tyGen.tyBtnTeachBtmPos2.bRtCompl = TRUE THEN
		tyP1021McSetGen.tyGen.tyBtnTeachBtmPos2.bRtCompl		:= FALSE;
		tyP1021McSetGen.tyGen.tyBtnTeachBtmPos2.bValue		:= FALSE;

		bTeachLifterBtmPos2	:= TRUE;
		eChgPage			:= UIP1026McSetTeach;

	END_IF

END_ACTION
```

#### Act_OptP1021Keypad.st
```iecst
ACTION Act_OptP1021Keypad:

	IF fUIOutRtStatTPIsOpen(ADR(tyP1021McSetGen.tyGen.tyStringMcNm.uiRtStat)) = TRUE THEN
		tyProperty.tyKeypad.tyStringTitle.sKeypadTitle	:= tyP1021McSetGen.tyGen.tyStringMcNm.sKeypadTitle;

	ELSIF fUIOutRtStatTPIsOpen(ADR(tyP1021McSetGen.tyGen.tyNumSSaverTm.uiRtStat)) = TRUE THEN
		tyProperty.tyKeypad.tyStringTitle.sKeypadTitle	:= tyP1021McSetGen.tyGen.tyNumSSaverTm.sKeypadTitle;

	ELSIF fUIOutRtStatTPIsOpen(ADR(tyP1021McSetGen.tyGen.tyStringIPAddr.uiRtStat)) = TRUE THEN
		tyProperty.tyKeypad.tyStringTitle.sKeypadTitle	:= tyP1021McSetGen.tyGen.tyStringIPAddr.sKeypadTitle;

	ELSIF fUIOutRtStatTPIsOpen(ADR(tyP1021McSetGen.tyGen.tyStringSubnetMask.uiRtStat)) = TRUE THEN
		tyProperty.tyKeypad.tyStringTitle.sKeypadTitle	:= tyP1021McSetGen.tyGen.tyStringSubnetMask.sKeypadTitle;
		//ADD
	ELSIF fUIOutRtStatTPIsOpen(ADR(tyP1021McSetGen.tyGen.tyStringHMIIPAddr.uiRtStat)) = TRUE THEN
		tyProperty.tyKeypad.tyTxtTitle.sTxt		:= tyP1021McSetGen.tyGen.tyStringHMIIPAddr.sKeypadTitle;

	ELSIF fUIOutRtStatTPIsOpen(ADR(tyP1021McSetGen.tyGen.tyNumConvInitTm.uiRtStat)) = TRUE THEN
		tyProperty.tyKeypad.tyStringTitle.sKeypadTitle	:= tyP1021McSetGen.tyGen.tyNumConvInitTm.sKeypadTitle;

	ELSIF fUIOutRtStatTPIsOpen(ADR(tyP1021McSetGen.tyGen.tyNumWidthAtHm.uiRtStat)) = TRUE THEN
		tyProperty.tyKeypad.tyStringTitle.sKeypadTitle	:= tyP1021McSetGen.tyGen.tyNumWidthAtHm.sKeypadTitle;

	ELSIF fUIOutRtStatTPIsOpen(ADR(tyP1021McSetGen.tyGen.tyNumTranInErrDlyTm.uiRtStat)) = TRUE THEN
		tyProperty.tyKeypad.tyStringTitle.sKeypadTitle	:= tyP1021McSetGen.tyGen.tyNumTranInErrDlyTm.sKeypadTitle;

	ELSIF fUIOutRtStatTPIsOpen(ADR(tyP1021McSetGen.tyGen.tyNumMag1ConvRunTm.uiRtStat)) = TRUE THEN
		tyProperty.tyKeypad.tyStringTitle.sKeypadTitle	:= tyP1021McSetGen.tyGen.tyNumMag1ConvRunTm.sKeypadTitle;

	ELSIF fUIOutRtStatTPIsOpen(ADR(tyP1021McSetGen.tyGen.tyNumMag2ConvRunTm.uiRtStat)) = TRUE THEN
		tyProperty.tyKeypad.tyStringTitle.sKeypadTitle	:= tyP1021McSetGen.tyGen.tyNumMag2ConvRunTm.sKeypadTitle;

	ELSIF fUIOutRtStatTPIsOpen(ADR(tyP1021McSetGen.tyGen.tyNumMag3ConvRunTm.uiRtStat)) = TRUE THEN
		tyProperty.tyKeypad.tyStringTitle.sKeypadTitle	:= tyP1021McSetGen.tyGen.tyNumMag3ConvRunTm.sKeypadTitle;

	ELSIF fUIOutRtStatTPIsOpen(ADR(tyP1021McSetGen.tyGen.tyNumTravPosLaneA.uiRtStat)) = TRUE THEN
		tyProperty.tyKeypad.tyStringTitle.sKeypadTitle	:= tyP1021McSetGen.tyGen.tyNumTravPosLaneA.sKeypadTitle;

	ELSIF fUIOutRtStatTPIsOpen(ADR(tyP1021McSetGen.tyGen.tyNumTravPosLaneB.uiRtStat)) = TRUE THEN
		tyProperty.tyKeypad.tyStringTitle.sKeypadTitle	:= tyP1021McSetGen.tyGen.tyNumTravPosLaneB.sKeypadTitle;

	ELSIF fUIOutRtStatTPIsOpen(ADR(tyP1021McSetGen.tyGen.tyNumLiftPosLaneA.uiRtStat)) = TRUE THEN
		tyProperty.tyKeypad.tyStringTitle.sKeypadTitle	:= tyP1021McSetGen.tyGen.tyNumLiftPosLaneA.sKeypadTitle;

	ELSIF fUIOutRtStatTPIsOpen(ADR(tyP1021McSetGen.tyGen.tyNumLiftPosLaneB.uiRtStat)) = TRUE THEN
		tyProperty.tyKeypad.tyStringTitle.sKeypadTitle	:= tyP1021McSetGen.tyGen.tyNumLiftPosLaneB.sKeypadTitle;

	ELSIF fUIOutRtStatTPIsOpen(ADR(tyP1021McSetGen.tyGen.tyNumWidthOffset.uiRtStat)) = TRUE THEN
		tyProperty.tyKeypad.tyStringTitle.sKeypadTitle	:= tyP1021McSetGen.tyGen.tyNumWidthOffset.sKeypadTitle;

	ELSIF fUIOutRtStatTPIsOpen(ADR(tyP1021McSetGen.tyGen.tyNumAutoLogoutTm.uiRtStat)) = TRUE THEN
		tyProperty.tyKeypad.tyStringTitle.sKeypadTitle	:= tyP1021McSetGen.tyGen.tyNumAutoLogoutTm.sKeypadTitle;

	ELSIF fUIOutRtStatTPIsOpen(ADR(tyP1021McSetGen.tyNetwork.tyStringIPAddr.uiRtStat)) = TRUE THEN
		tyProperty.tyKeypad.tyStringTitle.sKeypadTitle	:= tyP1021McSetGen.tyNetwork.tyStringIPAddr.sKeypadTitle;

	ELSIF fUIOutRtStatTPIsOpen(ADR(tyP1021McSetGen.tyNetwork.tyStringSubnetMask.uiRtStat)) = TRUE THEN
		tyProperty.tyKeypad.tyStringTitle.sKeypadTitle	:= tyP1021McSetGen.tyNetwork.tyStringSubnetMask.sKeypadTitle;

	ELSIF fUIOutRtStatTPIsOpen(ADR(tyP1021McSetGen.tyGen.tyNumMagAutoDetSenTm.uiRtStat)) = TRUE THEN
		tyProperty.tyKeypad.tyStringTitle.sKeypadTitle	:= tyP1021McSetGen.tyGen.tyNumMagAutoDetSenTm.sKeypadTitle;

	ELSIF fUIOutRtStatTPIsOpen(ADR(tyP1021McSetGen.tyGen.tyNumMag1WidthAtHm.uiRtStat)) = TRUE THEN
		tyProperty.tyKeypad.tyStringTitle.sKeypadTitle	:= tyP1021McSetGen.tyGen.tyNumMag1WidthAtHm.sKeypadTitle;

	ELSIF fUIOutRtStatTPIsOpen(ADR(tyP1021McSetGen.tyGen.tyNumMag2WidthAtHm.uiRtStat)) = TRUE THEN
		tyProperty.tyKeypad.tyStringTitle.sKeypadTitle	:= tyP1021McSetGen.tyGen.tyNumMag2WidthAtHm.sKeypadTitle;

	ELSIF fUIOutRtStatTPIsOpen(ADR(tyP1021McSetGen.tyGen.tyNumMag3WidthAtHm.uiRtStat)) = TRUE THEN
		tyProperty.tyKeypad.tyStringTitle.sKeypadTitle	:= tyP1021McSetGen.tyGen.tyNumMag3WidthAtHm.sKeypadTitle;

	ELSIF fUIOutRtStatTPIsOpen(ADR(tyP1021McSetGen.tyGen.tyNumAutoLogoutTm.uiRtStat)) = TRUE THEN
		tyProperty.tyKeypad.tyStringTitle.sKeypadTitle	:= tyP1021McSetGen.tyGen.tyNumAutoLogoutTm.sKeypadTitle;

	ELSIF fUIOutRtStatTPIsOpen(ADR(tyP1021McSetGen.tyGen.tyNumAWPusherAtHm.uiRtStat)) = TRUE THEN
		tyProperty.tyKeypad.tyStringTitle.sKeypadTitle	:= tyP1021McSetGen.tyGen.tyNumAWPusherAtHm.sKeypadTitle;

	ELSIF fUIOutRtStatTPIsOpen(ADR(tyP1021McSetGen.tyGen.tyNumTravFixtoFixPosInlet.uiRtStat)) = TRUE THEN
		tyProperty.tyKeypad.tyStringTitle.sKeypadTitle	:= tyP1021McSetGen.tyGen.tyNumTravFixtoFixPosInlet.sKeypadTitle;

	ELSIF fUIOutRtStatTPIsOpen(ADR(tyP1021McSetGen.tyGen.tyNumTCPSvrPort.uiRtStat)) = TRUE THEN
		tyProperty.tyKeypad.tyStringTitle.sKeypadTitle	:= tyP1021McSetGen.tyGen.tyNumTCPSvrPort.sKeypadTitle;

	ELSIF fUIOutRtStatTPIsOpen(ADR(tyP1021McSetGen.tyGen.tyNumMag1WidthChkDetDist.uiRtStat)) = TRUE THEN
		tyProperty.tyKeypad.tyStringTitle.sKeypadTitle	:= tyP1021McSetGen.tyGen.tyNumMag1WidthChkDetDist.sKeypadTitle;

	ELSIF fUIOutRtStatTPIsOpen(ADR(tyP1021McSetGen.tyGen.tyNumMag2WidthChkDetDist.uiRtStat)) = TRUE THEN
		tyProperty.tyKeypad.tyStringTitle.sKeypadTitle	:= tyP1021McSetGen.tyGen.tyNumMag2WidthChkDetDist.sKeypadTitle;

	ELSIF fUIOutRtStatTPIsOpen(ADR(tyP1021McSetGen.tyGen.tyNumMag3WidthChkDetDist.uiRtStat)) = TRUE THEN
		tyProperty.tyKeypad.tyStringTitle.sKeypadTitle	:= tyP1021McSetGen.tyGen.tyNumMag3WidthChkDetDist.sKeypadTitle;

	ELSIF fUIOutRtStatTPIsOpen(ADR(tyP1021McSetGen.tyGen.tyStringDefaultGWIP.uiRtStat)) = TRUE THEN
		tyProperty.tyKeypad.tyStringTitle.sKeypadTitle	:= tyP1021McSetGen.tyGen.tyStringDefaultGWIP.sKeypadTitle;
	ELSE
		tyProperty.tyKeypad.tyStringTitle.sKeypadTitle	:= '';

	END_IF

END_ACTION
```

#### Act_OptP1021IPAddr.st
```iecst
ACTION Act_OptP1021IPAddr:

	IF tyP1021McSetGen.tyGen.tyStringIPAddr.bRtCompl = TRUE THEN

		IF fIPValid(tyP1021McSetGen.tyGen.tyStringIPAddr.sValue , ADR(a_iIPPart1)) THEN

			IF usiSaveIPAddrStep = 0 THEN
				p_tyC0008MsgBox ACCESS ADR(tyP1021McSetGen.tyMsgBoxUpdtIPAddrAsk);

				IF tyP1021McSetGen.tyMsgBoxUpdtIPAddrAsk.tyBtnYes.bRtCompl = TRUE THEN
					tyP1021McSetGen.tyMsgBoxUpdtIPAddrAsk.tyBtnYes.bRtCompl	:= FALSE;
					tyP1021McSetGen.tyMsgBoxUpdtIPAddrAsk.tyBtnYes.bValue	:= FALSE;

					p_tyC0008MsgBox ACCESS ADR(tyP1021McSetGen.tyMsgBoxHide);

					usiSaveIPAddrStep	:= 1;

				ELSIF tyP1021McSetGen.tyMsgBoxUpdtIPAddrAsk.tyBtnNo.bRtCompl = TRUE THEN
					tyP1021McSetGen.tyMsgBoxUpdtIPAddrAsk.tyBtnNo.bRtCompl	:= FALSE;
					tyP1021McSetGen.tyMsgBoxUpdtIPAddrAsk.tyBtnNo.bValue	:= FALSE;

					//Recover IP Address
					tyP1021McSetGen.tyGen.tyStringIPAddr.sValue	:= p_sHWInfoIPAddr;

					tyP1021McSetGen.tyGen.tyStringIPAddr.bRtCompl	:= FALSE;

					p_tyC0008MsgBox ACCESS ADR(tyP1021McSetGen.tyMsgBoxHide);

				END_IF

			ELSIF usiSaveIPAddrStep = 1 THEN
				//Set IP Address
				sSetIPAddr	:= tyP1021McSetGen.tyGen.tyStringIPAddr.sValue;

				eHWInfoAct	:= HWInfoActSetIPAddr;

				IF p_eHWInfoStat = HWInfoActSetIPAddr AND p_eHWInfoStatus = Done THEN
					eHWInfoAct	:= HWInfoActIdle;

					bUpdateP1021Network	:= TRUE;

					usiSaveIPAddrStep	:= 0;

					tyP1021McSetGen.tyGen.tyStringIPAddr.bRtCompl	:= FALSE;

				ELSIF p_eHWInfoStatus = Error THEN
					p_tyC0008MsgBox ACCESS ADR(tyP1021McSetGen.tyMsgBoxUpdtIPAddrErr);

					IF tyP1021McSetGen.tyMsgBoxUpdtIPAddrErr.tyBtnNo.bRtCompl = TRUE THEN
						tyP1021McSetGen.tyMsgBoxUpdtIPAddrErr.tyBtnNo.bRtCompl	:= FALSE;
						tyP1021McSetGen.tyMsgBoxUpdtIPAddrErr.tyBtnNo.bValue	:= FALSE;

						p_tyC0008MsgBox ACCESS ADR(tyP1021McSetGen.tyMsgBoxHide);

						//Recover IP Address
						tyP1021McSetGen.tyGen.tyStringIPAddr.sValue	:= p_sHWInfoIPAddr;

						usiSaveIPAddrStep	:= 0;

						tyP1021McSetGen.tyGen.tyStringIPAddr.bRtCompl	:= FALSE;

					END_IF

				END_IF

			END_IF

		ELSE

			p_tyC0008MsgBox ACCESS ADR(tyP1021McSetGen.tyMsgBoxIPAddrInvalid);

			IF tyP1021McSetGen.tyMsgBoxIPAddrInvalid.tyBtnNo.bRtCompl = TRUE THEN
				tyP1021McSetGen.tyMsgBoxIPAddrInvalid.tyBtnNo.bRtCompl	:= FALSE;
				tyP1021McSetGen.tyMsgBoxIPAddrInvalid.tyBtnNo.bValue	:= FALSE;

				p_tyC0008MsgBox ACCESS ADR(tyP1021McSetGen.tyMsgBoxHide);

				//Recover IP Address
				tyP1021McSetGen.tyGen.tyStringIPAddr.sValue	:= p_sHWInfoIPAddr;

				tyP1021McSetGen.tyGen.tyStringIPAddr.bRtCompl	:= FALSE;

			END_IF

		END_IF

	END_IF

END_ACTION
```

#### Act_OptP1021SubnetMask.st
```iecst
ACTION Act_OptP1021SubnetMask:

	IF tyP1021McSetGen.tyGen.tyStringSubnetMask.bRtCompl = TRUE THEN

		IF fIPValid(tyP1021McSetGen.tyGen.tyStringSubnetMask.sValue , ADR(a_iSubnetMaskPart1)) THEN

			IF usiSaveSubnetMaskStep = 0 THEN
				p_tyC0008MsgBox ACCESS ADR(tyP1021McSetGen.tyMsgBoxUpdtSubnetAsk);

				IF tyP1021McSetGen.tyMsgBoxUpdtSubnetAsk.tyBtnYes.bRtCompl = TRUE THEN
					tyP1021McSetGen.tyMsgBoxUpdtSubnetAsk.tyBtnYes.bRtCompl	:= FALSE;
					tyP1021McSetGen.tyMsgBoxUpdtSubnetAsk.tyBtnYes.bValue	:= FALSE;

					p_tyC0008MsgBox ACCESS ADR(tyP1021McSetGen.tyMsgBoxHide);

					usiSaveSubnetMaskStep	:= 1;

				ELSIF tyP1021McSetGen.tyMsgBoxUpdtSubnetAsk.tyBtnNo.bRtCompl = TRUE THEN
					tyP1021McSetGen.tyMsgBoxUpdtSubnetAsk.tyBtnNo.bRtCompl	:= FALSE;
					tyP1021McSetGen.tyMsgBoxUpdtSubnetAsk.tyBtnNo.bValue	:= FALSE;

					p_tyC0008MsgBox ACCESS ADR(tyP1021McSetGen.tyMsgBoxHide);

					//Recover Subnet Mask
					tyP1021McSetGen.tyGen.tyStringSubnetMask.sValue	:= p_sHWInfoSubnetMask;

					tyP1021McSetGen.tyGen.tyStringSubnetMask.bRtCompl	:= FALSE;

				END_IF

			ELSIF usiSaveSubnetMaskStep = 1 THEN
				//Set Subnet Mask
				sSetSubnetMask	:= tyP1021McSetGen.tyGen.tyStringSubnetMask.sValue;

				eHWInfoAct	:= HWInfoActSetSubnetMask;

				IF p_eHWInfoStat = HWInfoActSetSubnetMask AND p_eHWInfoStatus = Done THEN
					eHWInfoAct	:= HWInfoActIdle;

					bUpdateP1021Network	:= TRUE;

					usiSaveSubnetMaskStep	:= 0;

					tyP1021McSetGen.tyGen.tyStringSubnetMask.bRtCompl	:= FALSE;

				ELSIF p_eHWInfoStatus = Error THEN
					p_tyC0008MsgBox ACCESS ADR(tyP1021McSetGen.tyMsgBoxUpdtSubnetErr);

					IF tyP1021McSetGen.tyMsgBoxUpdtSubnetErr.tyBtnNo.bRtCompl = TRUE THEN
						tyP1021McSetGen.tyMsgBoxUpdtSubnetErr.tyBtnNo.bRtCompl	:= FALSE;
						tyP1021McSetGen.tyMsgBoxUpdtSubnetErr.tyBtnNo.bValue	:= FALSE;

						p_tyC0008MsgBox ACCESS ADR(tyP1021McSetGen.tyMsgBoxHide);

						//Recover Subnet Mask
						tyP1021McSetGen.tyGen.tyStringSubnetMask.sValue	:= p_sHWInfoSubnetMask;

						usiSaveSubnetMaskStep	:= 0;

						tyP1021McSetGen.tyGen.tyStringSubnetMask.bRtCompl	:= FALSE;

					END_IF

				END_IF

			END_IF

		ELSE

			p_tyC0008MsgBox ACCESS ADR(tyP1021McSetGen.tyMsgBoxSubnetInvalid);

			IF tyP1021McSetGen.tyMsgBoxSubnetInvalid.tyBtnNo.bRtCompl = TRUE THEN
				tyP1021McSetGen.tyMsgBoxSubnetInvalid.tyBtnNo.bRtCompl	:= FALSE;
				tyP1021McSetGen.tyMsgBoxSubnetInvalid.tyBtnNo.bValue	:= FALSE;

				p_tyC0008MsgBox ACCESS ADR(tyP1021McSetGen.tyMsgBoxHide);

				//Recover Subnet Mask
				tyP1021McSetGen.tyGen.tyStringSubnetMask.sValue	:= p_sHWInfoSubnetMask;

				tyP1021McSetGen.tyGen.tyStringSubnetMask.bRtCompl	:= FALSE;

			END_IF

		END_IF

	END_IF

END_ACTION
```

#### Act_OptP1021DHCPSetting.st
```iecst
ACTION Act_OptP1021DHCPSetting:

	IF p_tyMcParamCurr.eNetworkMod = IPFromDHCPServer  THEN
		fUIInRtStatOff(ADR(tyP1021McSetGen.tyGen.tyStringIPAddr.uiMaskRtStat));
		fUIInRtStatOff(ADR(tyP1021McSetGen.tyGen.tyStringSubnetMask.uiMaskRtStat));
	ELSE
		fUIInRtStatHide(ADR(tyP1021McSetGen.tyGen.tyStringIPAddr.uiMaskRtStat));
		fUIInRtStatHide(ADR(tyP1021McSetGen.tyGen.tyStringSubnetMask.uiMaskRtStat));
	END_IF

	//Trigger Save Condition
	IF tyP1021McSetGen.tyGen.tyDrpDnNetworkMod.bRtCompl THEN

		bSaveNetworkPriority := TRUE;

		usiNetworkModeNew := tyP1021McSetGen.tyGen.tyDrpDnNetworkMod.usiValueIdx;

		fUIInRtStatHide(ADR(tyCommon.tySet.tyBtnSave.uiMaskRtStat));

		tyP1021McSetGen.tyGen.tyDrpDnNetworkMod.bRtCompl := FALSE;

		IF usiNetworkModeOld<>usiNetworkModeNew THEN
			IF tyP1021McSetGen.tyGen.tyDrpDnNetworkMod.usiValueIdx = DINT_TO_USINT(SetIPManually) THEN

				tyP1021McSetGen.tyNetwork.tyStringIPAddr.sValue		:= p_sHWInfoIPAddr;
				tyP1021McSetGen.tyNetwork.tyStringSubnetMask.sValue	:= p_sHWInfoSubnetMask;
				fUIInRtStatOff(ADR(tyP1021McSetGen.tyNetwork.tyLyr.uiRtStat));

			END_IF
		END_IF

	END_IF

	// If Change from DHCP to Manual, Pop Up Detail to fill in
	IF tyP1021McSetGen.tyNetwork.tyLyr.uiRtStat.0 = FALSE THEN
		//IP Check
		IF tyP1021McSetGen.tyNetwork.tyStringIPAddr.bRtCompl = TRUE THEN
			IF fIPValid(tyP1021McSetGen.tyNetwork.tyStringIPAddr.sValue , ADR(a_iIPPart1)) THEN

				tyP1021McSetGen.tyNetwork.tyStringIPAddr.bRtCompl	:= FALSE;
			ELSE
				p_tyC0008MsgBox ACCESS ADR(tyP1021McSetGen.tyMsgBoxIPAddrInvalidEdit);

				IF tyP1021McSetGen.tyMsgBoxIPAddrInvalidEdit.tyBtnNo.bRtCompl = TRUE THEN
					tyP1021McSetGen.tyMsgBoxIPAddrInvalidEdit.tyBtnNo.bRtCompl	:= FALSE;
					tyP1021McSetGen.tyMsgBoxIPAddrInvalidEdit.tyBtnNo.bValue	:= FALSE;

					p_tyC0008MsgBox ACCESS ADR(tyP1021McSetGen.tyMsgBoxHide);

					//Recover IP Address
					tyP1021McSetGen.tyNetwork.tyStringIPAddr.sValue	:= p_sHWInfoIPAddr;
					tyP1021McSetGen.tyNetwork.tyStringIPAddr.bRtCompl	:= FALSE;
				END_IF
			END_IF
		END_IF

		//Subnet Check
		IF tyP1021McSetGen.tyNetwork.tyStringSubnetMask.bRtCompl = TRUE THEN
			IF fIPValid(tyP1021McSetGen.tyNetwork.tyStringSubnetMask.sValue , ADR(a_iSubnetMaskPart1)) THEN

				tyP1021McSetGen.tyNetwork.tyStringSubnetMask.bRtCompl	:= FALSE;
			ELSE
				p_tyC0008MsgBox ACCESS ADR(tyP1021McSetGen.tyMsgBoxSubnetInvalidEdit);

				IF tyP1021McSetGen.tyMsgBoxSubnetInvalidEdit.tyBtnNo.bRtCompl = TRUE THEN
					tyP1021McSetGen.tyMsgBoxSubnetInvalidEdit.tyBtnNo.bRtCompl	:= FALSE;
					tyP1021McSetGen.tyMsgBoxSubnetInvalidEdit.tyBtnNo.bValue	:= FALSE;

					p_tyC0008MsgBox ACCESS ADR(tyP1021McSetGen.tyMsgBoxHide);
					//Recover IP Address
					tyP1021McSetGen.tyNetwork.tyStringSubnetMask.sValue	:= p_sHWInfoSubnetMask;
					tyP1021McSetGen.tyNetwork.tyStringSubnetMask.bRtCompl	:= FALSE;

				END_IF
			END_IF
		END_IF

		IF tyP1021McSetGen.tyNetwork.tyBtnSave.bRtCompl = TRUE THEN

			tyP1021McSetGen.tyNetwork.tyBtnSave.bRtCompl	:= FALSE;
			tyP1021McSetGen.tyNetwork.tyBtnSave.bValue		:= FALSE;

			tyP1021McSetGen.tyGen.tyStringIPAddr.sValue 	:= tyP1021McSetGen.tyNetwork.tyStringIPAddr.sValue;
			tyP1021McSetGen.tyGen.tyStringSubnetMask.sValue := tyP1021McSetGen.tyNetwork.tyStringSubnetMask.sValue;

			fUIInRtStatHide(ADR(tyP1021McSetGen.tyNetwork.tyLyr.uiRtStat));

		ELSIF tyP1021McSetGen.tyNetwork.tyBtnCancel.bRtCompl = TRUE THEN
			tyP1021McSetGen.tyNetwork.tyBtnCancel.bRtCompl	:= FALSE;
			tyP1021McSetGen.tyNetwork.tyBtnCancel.bValue	:= FALSE;

			fUIInRtStatHide(ADR(tyP1021McSetGen.tyNetwork.tyLyr.uiRtStat));

		END_IF

	END_IF

	//Once click save, change config
	IF tyCommon.tySet.tyBtnSave.bRtCompl = TRUE AND bSaveNetworkPriority AND NOT bNetworkConfigChanged THEN

		IF usiNetworkModeOld<>usiNetworkModeNew THEN

			IF usiChgNetworkConfigStep = 0 THEN

				IF usiNetworkModeNew = DINT_TO_USINT(IPFromDHCPServer) THEN
					tyP1021McSetGen.tyMsgBoxChgNetworkAsk.tyTxtMsg.usiValueIdx := 109;
				ELSE
					tyP1021McSetGen.tyMsgBoxChgNetworkAsk.tyTxtMsg.usiValueIdx := 110;
				END_IF

				p_tyC0008MsgBox ACCESS ADR(tyP1021McSetGen.tyMsgBoxChgNetworkAsk);

				IF tyP1021McSetGen.tyMsgBoxChgNetworkAsk.tyBtnYes.bRtCompl = TRUE THEN
					tyP1021McSetGen.tyMsgBoxChgNetworkAsk.tyBtnYes.bRtCompl	:= FALSE;
					tyP1021McSetGen.tyMsgBoxChgNetworkAsk.tyBtnYes.bValue	:= FALSE;

					p_tyC0008MsgBox ACCESS ADR(tyP1021McSetGen.tyMsgBoxHide);

					usiChgNetworkConfigStep	:= 1;

				ELSIF tyP1021McSetGen.tyMsgBoxChgNetworkAsk.tyBtnNo.bRtCompl = TRUE THEN
					tyP1021McSetGen.tyMsgBoxChgNetworkAsk.tyBtnNo.bRtCompl	:= FALSE;
					tyP1021McSetGen.tyMsgBoxChgNetworkAsk.tyBtnNo.bValue	:= FALSE;

					tyP1021McSetGen.tyGen.tyStringIPAddr.sValue		:= p_sHWInfoIPAddr;
					tyP1021McSetGen.tyGen.tyStringSubnetMask.sValue := p_sHWInfoSubnetMask;

					//Recover Old Dropdown Value
					tyP1021McSetGen.tyGen.tyDrpDnNetworkMod.usiValueIdx	:= usiNetworkModeOld;

					//Reset Save Priority
					bSaveNetworkPriority := FALSE;

					//Reset Network Step
					usiChgNetworkConfigStep	:= 0;

					p_tyC0008MsgBox ACCESS ADR(tyP1021McSetGen.tyMsgBoxHide);

				END_IF

			ELSIF usiChgNetworkConfigStep = 1 THEN

				IF usiNetworkModeNew = DINT_TO_USINT(IPFromDHCPServer) THEN
					usiNetworkModeSelected := DINT_TO_USINT(IPFromDHCPServer);
				ELSE
					usiNetworkModeSelected := DINT_TO_USINT(SetIPManually);
				END_IF

				eHWInfoAct	:= HWInfoActSetEthConfigMode;

				IF p_eHWInfoStat = HWInfoActSetEthConfigMode AND p_eHWInfoStatus = Done THEN
					eHWInfoAct	:= HWInfoActIdle;

					usiChgNetworkConfigStep	:= 2;

				ELSIF p_eHWInfoStatus = Error THEN
					p_tyC0008MsgBox ACCESS ADR(tyP1021McSetGen.tyMsgBoxSetDHCPError);

					IF tyP1021McSetGen.tyMsgBoxSetDHCPError.tyBtnNo.bRtCompl = TRUE THEN
						tyP1021McSetGen.tyMsgBoxSetDHCPError.tyBtnNo.bRtCompl	:= FALSE;
						tyP1021McSetGen.tyMsgBoxSetDHCPError.tyBtnNo.bValue	:= FALSE;

						p_tyC0008MsgBox ACCESS ADR(tyP1021McSetGen.tyMsgBoxHide);

						//Recover Old Dropdown Value
						tyP1021McSetGen.tyGen.tyDrpDnNetworkMod.usiValueIdx	:= usiNetworkModeOld;

						//Reset Network Step
						usiChgNetworkConfigStep	:= 0;

						//Reset Save Priority
						bSaveNetworkPriority := FALSE;

					END_IF
				END_IF

			ELSIF usiChgNetworkConfigStep = 2 THEN

				IF p_eHWInfoStat = HWInfoActIdle THEN

					usiChgNetworkConfigStep := 0;
					bNetworkConfigChanged := TRUE;

				END_IF

			END_IF

		ELSE
			//Reset Save Priority
			bSaveNetworkPriority := FALSE;
		END_IF

	END_IF

	//Refresh/Set IP Address and Subnet Mask
	IF bNetworkConfigChanged THEN

		IF usiRefreshDetailStep = 0 THEN
			IF usiNetworkModeNew = DINT_TO_USINT(IPFromDHCPServer) THEN

				eHWInfoAct	:= HWInfoActGetIPAddr;

				IF p_eHWInfoStat = HWInfoActGetIPAddr AND p_eHWInfoStatus = Done THEN
					eHWInfoAct	:= HWInfoActIdle;

					usiRefreshDetailStep	:= 1;

					//Refresh IP value
					tyP1021McSetGen.tyGen.tyStringIPAddr.sValue := p_sHWInfoIPAddr;

				ELSIF p_eHWInfoStatus = Error THEN
					p_tyC0008MsgBox ACCESS ADR(tyP1021McSetGen.tyMsgBoxGetIPAddrErr);

					IF tyP1021McSetGen.tyMsgBoxGetIPAddrErr.tyBtnNo.bRtCompl = TRUE THEN
						tyP1021McSetGen.tyMsgBoxGetIPAddrErr.tyBtnNo.bRtCompl	:= FALSE;
						tyP1021McSetGen.tyMsgBoxGetIPAddrErr.tyBtnNo.bValue	:= FALSE;

						p_tyC0008MsgBox ACCESS ADR(tyP1021McSetGen.tyMsgBoxHide);

						//Reset Save Priority
						bSaveNetworkPriority := FALSE;

						//Reset Refresh Step
						usiRefreshDetailStep	:= 0;

						bNetworkConfigChanged	:= FALSE;

					END_IF
				END_IF

			ELSE
				eHWInfoAct	:= HWInfoActSetIPAddr;

				sSetIPAddr	:= tyP1021McSetGen.tyGen.tyStringIPAddr.sValue;

				IF p_eHWInfoStat = HWInfoActSetIPAddr AND p_eHWInfoStatus = Done THEN
					eHWInfoAct	:= HWInfoActIdle;

					usiRefreshDetailStep	:= 1;

				ELSIF p_eHWInfoStatus = Error THEN
					p_tyC0008MsgBox ACCESS ADR(tyP1021McSetGen.tyMsgBoxUpdtIPAddrErr);

					IF tyP1021McSetGen.tyMsgBoxUpdtIPAddrErr.tyBtnNo.bRtCompl = TRUE THEN
						tyP1021McSetGen.tyMsgBoxUpdtIPAddrErr.tyBtnNo.bRtCompl	:= FALSE;
						tyP1021McSetGen.tyMsgBoxUpdtIPAddrErr.tyBtnNo.bValue	:= FALSE;

						p_tyC0008MsgBox ACCESS ADR(tyP1021McSetGen.tyMsgBoxHide);

						tyP1021McSetGen.tyGen.tyStringIPAddr.sValue := p_sHWInfoIPAddr;

						//Reset Save Priority
						bSaveNetworkPriority := FALSE;

						//Reset Refresh Step
						usiRefreshDetailStep	:= 0;

						bNetworkConfigChanged	:= FALSE;

					END_IF
				END_IF
			END_IF

		ELSIF usiRefreshDetailStep = 1 THEN

			IF p_eHWInfoStat = HWInfoActIdle THEN
				usiRefreshDetailStep := 2;
			END_IF

		ELSIF usiRefreshDetailStep = 2 THEN
			IF usiNetworkModeNew = DINT_TO_USINT(IPFromDHCPServer) THEN

				eHWInfoAct	:= HWInfoActGetSubnetMask;

				IF p_eHWInfoStat = HWInfoActGetSubnetMask AND p_eHWInfoStatus = Done THEN
					eHWInfoAct	:= HWInfoActIdle;

					//Reset Save Priority
					bSaveNetworkPriority := FALSE;

					//Reset Refresh Step
					usiRefreshDetailStep	:= 0;

					//Refresh subnet value
					tyP1021McSetGen.tyGen.tyStringSubnetMask.sValue := p_sHWInfoSubnetMask;

					bNetworkConfigChanged	:= FALSE;

				ELSIF p_eHWInfoStatus = Error THEN
					p_tyC0008MsgBox ACCESS ADR(tyP1021McSetGen.tyMsgBoxGetSubnetErr);

					IF tyP1021McSetGen.tyMsgBoxGetSubnetErr.tyBtnNo.bRtCompl = TRUE THEN
						tyP1021McSetGen.tyMsgBoxGetSubnetErr.tyBtnNo.bRtCompl	:= FALSE;
						tyP1021McSetGen.tyMsgBoxGetSubnetErr.tyBtnNo.bValue	:= FALSE;

						p_tyC0008MsgBox ACCESS ADR(tyP1021McSetGen.tyMsgBoxHide);

						//Reset Save Priority
						bSaveNetworkPriority := FALSE;

						//Reset Refresh Step
						usiRefreshDetailStep	:= 0;

						bNetworkConfigChanged	:= FALSE;

					END_IF
				END_IF

			ELSE
				eHWInfoAct	:= HWInfoActSetSubnetMask;

				sSetSubnetMask	:= tyP1021McSetGen.tyGen.tyStringSubnetMask.sValue;

				IF p_eHWInfoStat = HWInfoActSetSubnetMask AND p_eHWInfoStatus = Done THEN
					eHWInfoAct	:= HWInfoActIdle;

					//Reset Save Priority
					bSaveNetworkPriority := FALSE;

					//Reset Refresh Step
					usiRefreshDetailStep	:= 0;

					bNetworkConfigChanged	:= FALSE;

				ELSIF p_eHWInfoStatus = Error THEN
					p_tyC0008MsgBox ACCESS ADR(tyP1021McSetGen.tyMsgBoxUpdtSubnetErr);

					IF tyP1021McSetGen.tyMsgBoxUpdtSubnetErr.tyBtnNo.bRtCompl = TRUE THEN
						tyP1021McSetGen.tyMsgBoxUpdtSubnetErr.tyBtnNo.bRtCompl	:= FALSE;
						tyP1021McSetGen.tyMsgBoxUpdtSubnetErr.tyBtnNo.bValue	:= FALSE;

						p_tyC0008MsgBox ACCESS ADR(tyP1021McSetGen.tyMsgBoxHide);

						tyP1021McSetGen.tyGen.tyStringSubnetMask.sValue := p_sHWInfoSubnetMask;

						//Reset Save Priority
						bSaveNetworkPriority := FALSE;

						//Reset Refresh Step
						usiRefreshDetailStep	:= 0;

						bNetworkConfigChanged	:= FALSE;

					END_IF
				END_IF
			END_IF

		END_IF
	END_IF

END_ACTION
```

#### Act_OptP1021HMIIPAddr.st
```iecst
ACTION Act_OptP1021HMIIPAddr:

	IF tyP1021McSetGen.tyGen.tyStringHMIIPAddr.bRtCompl = TRUE THEN

		IF fIPValid(tyP1021McSetGen.tyGen.tyStringHMIIPAddr.sValue , ADR(a_iIPPart1)) THEN

			IF usiSaveHMIIPAddrStep = 0 THEN
				p_tyC0008MsgBox ACCESS ADR(tyP1021McSetGen.tyMsgBoxUpdtHMIIPAddrAsk);

				IF tyP1021McSetGen.tyMsgBoxUpdtHMIIPAddrAsk.tyBtnYes.bRtCompl = TRUE THEN
					tyP1021McSetGen.tyMsgBoxUpdtHMIIPAddrAsk.tyBtnYes.bRtCompl	:= FALSE;
					tyP1021McSetGen.tyMsgBoxUpdtHMIIPAddrAsk.tyBtnYes.bValue	:= FALSE;

					p_tyC0008MsgBox ACCESS ADR(tyP1021McSetGen.tyMsgBoxHide);

					usiSaveHMIIPAddrStep	:= 1;

				ELSIF tyP1021McSetGen.tyMsgBoxUpdtHMIIPAddrAsk.tyBtnNo.bRtCompl = TRUE THEN
					tyP1021McSetGen.tyMsgBoxUpdtHMIIPAddrAsk.tyBtnNo.bRtCompl	:= FALSE;
					tyP1021McSetGen.tyMsgBoxUpdtHMIIPAddrAsk.tyBtnNo.bValue	:= FALSE;

					//Recover IP Address
					tyP1021McSetGen.tyGen.tyStringHMIIPAddr.sValue	:= p_tyMcParamCurr.sHMIIPAddr;

					tyP1021McSetGen.tyGen.tyStringHMIIPAddr.bRtCompl	:= FALSE;

					p_tyC0008MsgBox ACCESS ADR(tyP1021McSetGen.tyMsgBoxHide);

				END_IF

			ELSIF usiSaveHMIIPAddrStep = 1 THEN
				//Set HMI IP Address
				sSetHMIIPAddr	:= tyP1021McSetGen.tyGen.tyStringHMIIPAddr.sValue;

				bUpdateP1021Network	:= TRUE;
				bUpdtHMIIPAddr := TRUE;

				IF p_eMcParamStat = McParamActWrite AND p_eMcParamStatus = Done THEN

					bUpdtHMIIPAddr := FALSE;

					usiSaveHMIIPAddrStep	:= 0;

					tyP1021McSetGen.tyGen.tyStringHMIIPAddr.bRtCompl	:= FALSE;

				ELSIF p_eMcParamStatus = Error THEN
					p_tyC0008MsgBox ACCESS ADR(tyP1021McSetGen.tyMsgBoxUpdtHMIIPAddrErr);

					IF tyP1021McSetGen.tyMsgBoxUpdtHMIIPAddrErr.tyBtnNo.bRtCompl = TRUE THEN
						tyP1021McSetGen.tyMsgBoxUpdtHMIIPAddrErr.tyBtnNo.bRtCompl	:= FALSE;
						tyP1021McSetGen.tyMsgBoxUpdtHMIIPAddrErr.tyBtnNo.bValue	:= FALSE;

						p_tyC0008MsgBox ACCESS ADR(tyP1021McSetGen.tyMsgBoxHide);

						//Recover IP Address
						tyP1021McSetGen.tyGen.tyStringHMIIPAddr.sValue	:= p_tyMcParamCurr.sHMIIPAddr;

						usiSaveHMIIPAddrStep	:= 0;

						tyP1021McSetGen.tyGen.tyStringHMIIPAddr.bRtCompl	:= FALSE;

						bUpdtHMIIPAddr := FALSE;
					END_IF

				END_IF

			END_IF

		ELSE

			p_tyC0008MsgBox ACCESS ADR(tyP1021McSetGen.tyMsgBoxHMIIPAddrInvalid);

			IF tyP1021McSetGen.tyMsgBoxHMIIPAddrInvalid.tyBtnNo.bRtCompl = TRUE THEN
				tyP1021McSetGen.tyMsgBoxHMIIPAddrInvalid.tyBtnNo.bRtCompl	:= FALSE;
				tyP1021McSetGen.tyMsgBoxHMIIPAddrInvalid.tyBtnNo.bValue	:= FALSE;

				p_tyC0008MsgBox ACCESS ADR(tyP1021McSetGen.tyMsgBoxHide);

				//Recover IP Address
				tyP1021McSetGen.tyGen.tyStringHMIIPAddr.sValue	:= p_tyMcParamCurr.sHMIIPAddr;

				tyP1021McSetGen.tyGen.tyStringHMIIPAddr.bRtCompl	:= FALSE;

			END_IF

		END_IF

	END_IF

END_ACTION
```

#### Act_EntP1022Disp.st
```iecst
ACTION Act_EntP1022Disp:
	//Access Address
	//new for Hermes 1.3
	IF p_tyNtParamCurr.bLFPrep OR p_tyNtParamCurr.bLCSLFPrep OR p_tyNtParamCurr.bLCSReqRcpPrep OR p_tyNtParamCurr.bLCSManageRcpPrep OR p_tyNtParamCurr.bLCSLiveDatPrep
		OR p_tyNtParamCurr.bLFUsrSetPrep OR p_tyNtParamCurr.bLFUsrSetPrep OR  p_tyNtParamCurr.bUSWidthChkPrep OR p_tyNtParamCurr.bDSWidthChkPrep THEN
		bNaviLyr1 := TRUE;
	ELSE
		bNaviLyr1 := FALSE;
	END_IF

	IF (p_tyNtParamCurr.bHermesSvyPrep AND p_tyMcParamCurr.bHermesSvyEn)  THEN
		bNaviLyr2 := TRUE;
	ELSE
		bNaviLyr2 := FALSE;
	END_IF

	IF bNaviLyr1 AND NOT bNaviLyr2 THEN
		p_tyC0004Navi ACCESS ADR(tyP1022McSetVComm.tyNaviLyr1);
		fUIInRtStatOff(ADR(tyP1022McSetVComm.tyVComSel.tyLyr.uiRtStat)); //show
		fUIInRtStatHide(ADR(tyP1022McSetVComm.tyVComSvy.tyLyr.uiRtStat));
		fUIInRtStatOff(ADR(tyP1022McSetVComm.tyLF.tyLyr.uiRtStat)); //show

	ELSIF NOT bNaviLyr1 AND bNaviLyr2 THEN
		p_tyC0004Navi ACCESS ADR(tyP1022McSetVComm.tyNaviLyr2);
		fUIInRtStatHide(ADR(tyP1022McSetVComm.tyVComSel.tyLyr.uiRtStat)); //show
		fUIInRtStatOff(ADR(tyP1022McSetVComm.tyVComSvy.tyLyr.uiRtStat));
		fUIInRtStatHide(ADR(tyP1022McSetVComm.tyLF.tyLyr.uiRtStat)); //show

	ELSIF bNaviLyr1 AND bNaviLyr2 THEN
		p_tyC0004Navi ACCESS ADR(tyP1022McSetVComm.tyNaviLyr3);
		fUIInRtStatOff(ADR(tyP1022McSetVComm.tyVComSel.tyLyr.uiRtStat)); //show
		fUIInRtStatHide(ADR(tyP1022McSetVComm.tyVComSvy.tyLyr.uiRtStat));
		fUIInRtStatOff(ADR(tyP1022McSetVComm.tyLF.tyLyr.uiRtStat)); //show
	END_IF

	//Access Address
//	p_tyC0004Navi ACCESS ADR(tyP1022McSetVComm.tyNaviBack);

	p_tyC0005Main ACCESS ADR(tyCommon.tyMain);

	p_tyC0006Set ACCESS ADR(tyCommon.tySet);

	p_tyC0007Notif ACCESS ADR(tyCommon.tyNotif);

	p_tyC0008MsgBox ACCESS ADR(tyP1022McSetVComm.tyMsgBoxHide);

	p_tyC0009Info ACCESS ADR(tyCommon.tyInfo);

	p_tyP1022McSetVCommSel ACCESS ADR(tyP1022McSetVComm.tyVComSel);
	p_tyP1022McSetVCommLF ACCESS ADR(tyP1022McSetVComm.tyLF);
	p_tyP1022McSetVCommSvy ACCESS ADR(tyP1022McSetVComm.tyVComSvy); //new for Hermes 1.3

	//Backup Param
	tyP1022McSetVComm.tyVComSelBkUp	:= tyP1022McSetVComm.tyVComSel;
	tyP1022McSetVComm.tyLFBkUp		:= tyP1022McSetVComm.tyLF;
	tyP1022McSetVComm.tyVComSvyBkUp	:= tyP1022McSetVComm.tyVComSvy; //new for Hermes 1.3

END_ACTION
```

#### Act_OptP1022Navi.st
```iecst
ACTION Act_OptP1022Navi:

//	tyP1022McSetVComm.tyNaviBack.tyBtnBack.bRtLk	:= tyCommon.tySet.tyBtnSave.bRtCompl;
//
//	IF tyP1022McSetVComm.tyNaviBack.tyBtnBack.bRtCompl = TRUE THEN
//		eChgPage	:= UIP1020McSetNavi;
//
//		tyP1022McSetVComm.tyNaviBack.tyBtnBack.bRtCompl	:= FALSE;
//
//	END_IF

	tyP1022McSetVComm.tyNaviBack.tyBtnBack.bRtLk	:= tyCommon.tySet.tyBtnSave.bRtCompl;

	IF tyP1022McSetVComm.tyNaviLyr1.tyBtnBack.bRtCompl OR tyP1022McSetVComm.tyNaviLyr2.tyBtnBack.bRtCompl OR
		tyP1022McSetVComm.tyNaviLyr3.tyBtnBack.bRtCompl OR tyP1022McSetVComm.tyNaviLyr4.tyBtnBack.bRtCompl THEN
		tyP1022McSetVComm.tyNaviLyr1.tyBtnBack.bRtCompl	:= FALSE;
		tyP1022McSetVComm.tyNaviLyr2.tyBtnBack.bRtCompl	:= FALSE;
		tyP1022McSetVComm.tyNaviLyr3.tyBtnBack.bRtCompl	:= FALSE;
		tyP1022McSetVComm.tyNaviLyr4.tyBtnBack.bRtCompl	:= FALSE;

		eChgPage	:= UIP1020McSetNavi;

	ELSIF tyP1022McSetVComm.tyNaviLyr3.tyBtnLeft.bRtCompl = TRUE OR tyP1022McSetVComm.tyNaviLyr3.tyBtnRgt.bRtCompl = TRUE THEN
		tyP1022McSetVComm.tyNaviLyr3.tyBtnLeft.bRtCompl	:= FALSE;
		tyP1022McSetVComm.tyNaviLyr3.tyBtnRgt.bRtCompl	:= FALSE;

		p_tyC0004Navi ACCESS ADR(tyP1022McSetVComm.tyNaviLyr4);

		fUIInRtStatHide(ADR(tyP1022McSetVComm.tyVComSel.tyLyr.uiRtStat));
		fUIInRtStatOff(ADR(tyP1022McSetVComm.tyVComSvy.tyLyr.uiRtStat)); //new for Hermes 1.3
		fUIInRtStatHide(ADR(tyP1022McSetVComm.tyLF.tyLyr.uiRtStat));

	ELSIF tyP1022McSetVComm.tyNaviLyr4.tyBtnLeft.bRtCompl = TRUE OR tyP1022McSetVComm.tyNaviLyr4.tyBtnRgt.bRtCompl = TRUE THEN
		tyP1022McSetVComm.tyNaviLyr4.tyBtnLeft.bRtCompl	:= FALSE;
		tyP1022McSetVComm.tyNaviLyr4.tyBtnRgt.bRtCompl	:= FALSE;

		p_tyC0004Navi ACCESS ADR(tyP1022McSetVComm.tyNaviLyr3);

		fUIInRtStatOff(ADR(tyP1022McSetVComm.tyVComSel.tyLyr.uiRtStat));
		fUIInRtStatHide(ADR(tyP1022McSetVComm.tyVComSvy.tyLyr.uiRtStat));  //new for Hermes 1.3
		fUIInRtStatOff(ADR(tyP1022McSetVComm.tyLF.tyLyr.uiRtStat));
	END_IF

END_ACTION
```

#### Act_OptP1022Save.st
```iecst
ACTION Act_OptP1022Save:

	IF tyP1022McSetVComm.tyVComSel.tyBtnLF.bRtCompl 			OR tyP1022McSetVComm.tyVComSel.tyBtnLCSLF.bRtCompl
		OR tyP1022McSetVComm.tyVComSel.tyBtnLCSReqRcp.bRtCompl	OR tyP1022McSetVComm.tyVComSel.tyBtnLCSManageRcp.bRtCompl
		OR tyP1022McSetVComm.tyVComSel.tyBtnLCSLiveDat.bRtCompl	OR tyP1022McSetVComm.tyLF.tyBtnLeaderMc.bRtCompl
		OR tyP1022McSetVComm.tyLF.tyBtnSectionLdr.bRtCompl		OR tyP1022McSetVComm.tyLF.tyBtnUSWidthChkEn.bRtCompl
		OR tyP1022McSetVComm.tyLF.tyBtnSeqStayActive.bRtCompl OR tyP1022McSetVComm.tyLF.tyBtnDBAOnWOAlign.bRtCompl
		OR tyP1022McSetVComm.tyVComSvy.tyBtnConfiguration.bRtCompl OR tyP1022McSetVComm.tyVComSvy.tyBtnCheckAliveResponse.bRtCompl
		OR tyP1022McSetVComm.tyVComSvy.tyBtnBoardTracking.bRtCompl OR  tyP1022McSetVComm.tyVComSvy.tyBtnQueryWorkOrderInfo.bRtCompl
		OR 	tyP1022McSetVComm.tyVComSvy.tyBtnSendWorkOrderInfo.bRtCompl OR tyP1022McSetVComm.tyVComSvy.tyNumSndAliveTm.bRtCompl
		OR tyP1022McSetVComm.tyVComSvy.tyNumSvySystemPort.bRtCompl
	   	THEN

		fUIInRtStatHide(ADR(tyCommon.tySet.tyBtnSave.uiMaskRtStat));

		IF (NOT p_tyNtParamCurr.bLFUsrSetPrep AND NOT p_tyNtParamCurr.bLeaderMc) OR (p_tyNtParamCurr.bLFUsrSetPrep AND NOT tyP1022McSetVComm.tyLF.tyBtnLeaderMc.bValue) THEN
			IF tyP1022McSetVComm.tyVComSel.tyBtnLF.bRtCompl AND tyP1022McSetVComm.tyVComSel.tyBtnLF.bValue THEN
				tyP1022McSetVComm.tyVComSel.tyBtnLCSLF.bValue	:= FALSE;
			ELSIF tyP1022McSetVComm.tyVComSel.tyBtnLCSLF.bRtCompl AND tyP1022McSetVComm.tyVComSel.tyBtnLCSLF.bValue THEN
				tyP1022McSetVComm.tyVComSel.tyBtnLF.bValue		:= FALSE;
			END_IF

			IF tyP1022McSetVComm.tyVComSel.tyBtnLF.bValue = TRUE AND tyP1022McSetVComm.tyVComSel.tyBtnLCSLF.bValue = TRUE THEN
				tyP1022McSetVComm.tyVComSel.tyBtnLF.bValue		:= FALSE;
				tyP1022McSetVComm.tyVComSel.tyBtnLCSLF.bValue	:= FALSE;
			END_IF
		END_IF

		tyP1022McSetVComm.tyVComSel.tyBtnLF.bRtCompl			:= FALSE;
		tyP1022McSetVComm.tyVComSel.tyBtnLCSLF.bRtCompl			:= FALSE;
		tyP1022McSetVComm.tyVComSel.tyBtnLCSReqRcp.bRtCompl		:= FALSE;
		tyP1022McSetVComm.tyVComSel.tyBtnLCSManageRcp.bRtCompl	:= FALSE;
		tyP1022McSetVComm.tyVComSel.tyBtnLCSLiveDat.bRtCompl	:= FALSE;

		tyP1022McSetVComm.tyLF.tyBtnLeaderMc.bRtCompl			:= FALSE;
		tyP1022McSetVComm.tyLF.tyBtnSectionLdr.bRtCompl			:= FALSE;
		tyP1022McSetVComm.tyLF.tyBtnUSWidthChkEn.bRtCompl		:= FALSE;
		tyP1022McSetVComm.tyLF.tyBtnSeqStayActive.bRtCompl		:= FALSE;
		tyP1022McSetVComm.tyLF.tyBtnDBAOnWOAlign.bRtCompl		:= FALSE;

		//new for Hermes 1.3
		tyP1022McSetVComm.tyVComSvy.tyBtnConfiguration.bRtCompl			:= FALSE;
		tyP1022McSetVComm.tyVComSvy.tyBtnCheckAliveResponse.bRtCompl	:= FALSE;
		tyP1022McSetVComm.tyVComSvy.tyBtnBoardTracking.bRtCompl			:= FALSE;
		tyP1022McSetVComm.tyVComSvy.tyBtnQueryWorkOrderInfo.bRtCompl	:= FALSE;
		tyP1022McSetVComm.tyVComSvy.tyBtnSendWorkOrderInfo.bRtCompl		:= FALSE;
		tyP1022McSetVComm.tyVComSvy.tyNumSndAliveTm.bRtCompl			:= FALSE;
		tyP1022McSetVComm.tyVComSvy.tyNumSvySystemPort.bRtCompl			:= FALSE;

	END_IF

	IF tyCommon.tySet.tyBtnSave.bRtCompl = TRUE THEN

		tyMcParamWr.bLFEn			:=  tyP1022McSetVComm.tyVComSel.tyBtnLF.bValue;
		tyMcParamWr.bLCSLFEn		:=  tyP1022McSetVComm.tyVComSel.tyBtnLCSLF.bValue;
		tyMcParamWr.bLCSReqRcpEn	:=  tyP1022McSetVComm.tyVComSel.tyBtnLCSReqRcp.bValue;
		tyMcParamWr.bLCSManageRcpEn	:=  tyP1022McSetVComm.tyVComSel.tyBtnLCSManageRcp.bValue;
		tyMcParamWr.bLCSLiveDatEn	:=  tyP1022McSetVComm.tyVComSel.tyBtnLCSLiveDat.bValue;

		tyMcParamWr.bLFLeaderMc		:=	tyP1022McSetVComm.tyLF.tyBtnLeaderMc.bValue;
		tyMcParamWr.bSectionLeader	:=	tyP1022McSetVComm.tyLF.tyBtnSectionLdr.bValue;

		tyMcParamWr.bUSWidthChkEn	:=  tyP1022McSetVComm.tyLF.tyBtnUSWidthChkEn.bValue;
		tyMcParamWr.bLFSeqStayActive	:= 	tyP1022McSetVComm.tyLF.tyBtnSeqStayActive.bValue;
		tyMcParamWr.bDBAOnWOAlign		:= 	tyP1022McSetVComm.tyLF.tyBtnDBAOnWOAlign.bValue;

		//new for Hermes 1.3
		tyHermesSvyParamWr.bFeatureConfiguration	    	:=	tyP1022McSetVComm.tyVComSvy.tyBtnConfiguration.bValue;
		tyHermesSvyParamWr.bFeatureCheckAliveResponse		:=	tyP1022McSetVComm.tyVComSvy.tyBtnCheckAliveResponse.bValue;
		tyHermesSvyParamWr.bFeatureBoardTracking	    	:=	tyP1022McSetVComm.tyVComSvy.tyBtnBoardTracking.bValue;
		tyHermesSvyParamWr.bFeatureQueryWorkOrderInfo		:=	tyP1022McSetVComm.tyVComSvy.tyBtnQueryWorkOrderInfo.bValue;
		tyHermesSvyParamWr.bFeatureSendWorkOrderInfo		:=	tyP1022McSetVComm.tyVComSvy.tyBtnSendWorkOrderInfo.bValue;
		tyHermesSvyParamWr.tSndAlive		                :=	DINT_TO_TIME(tyP1022McSetVComm.tyVComSvy.tyNumSndAliveTm.diValue);
		tyHermesSvyParamWr.uiSvySvstemPort		            :=	DINT_TO_UINT(tyP1022McSetVComm.tyVComSvy.tyNumSvySystemPort.diValue);
		bSaveHMISvyConfig := TRUE;

		eMcParamAct	:= McParamActWrite;
		eHermesAct	:= HermesActWriteConfig; //new for Hermes 1.3

		IF p_eMcParamStat = McParamActWrite AND p_eMcParamStatus = Done THEN
			eMcParamAct	:= McParamActIdle;
			eHermesAct	:= HermesActIdle;  //new for Hermes 1.3

			//Update BackUp Param
			tyP1022McSetVComm.tyVComSelBkUp	:= tyP1022McSetVComm.tyVComSel;
			tyP1022McSetVComm.tyLFBkUp		:= tyP1022McSetVComm.tyLF;
			tyP1022McSetVComm.tyVComSvyBkUp	:= tyP1022McSetVComm.tyVComSvy;  //new for Hermes 1.3

			tyCommon.tySet.tyBtnSave.bRtCompl	:= FALSE;
			fUIInRtStatOff(ADR(tyCommon.tySet.tyBtnSave.uiMaskRtStat));
			bSaveHMISvyConfig := FALSE;  //new for Hermes 1.3

		ELSIF p_eMcParamStatus = Error THEN
			p_tyC0008MsgBox ACCESS ADR(tyP1022McSetVComm.tyMsgBoxSaveErr);

			IF tyP1022McSetVComm.tyMsgBoxSaveErr.tyBtnNo.bRtCompl = TRUE THEN
				tyP1022McSetVComm.tyMsgBoxSaveErr.tyBtnNo.bRtCompl 	:= FALSE;
				tyP1022McSetVComm.tyMsgBoxSaveErr.tyBtnNo.bValue	:= FALSE;

				p_tyC0008MsgBox ACCESS ADR(tyP1022McSetVComm.tyMsgBoxHide);

				//Restore Param
				tyP1022McSetVComm.tyVComSel	:= tyP1022McSetVComm.tyVComSelBkUp;
				tyP1022McSetVComm.tyVComSvy	:= tyP1022McSetVComm.tyVComSvyBkUp;  //new for Hermes 1.3
				tyP1022McSetVComm.tyLF		:= tyP1022McSetVComm.tyLFBkUp;
				tyMcParamWr					:= p_tyMcParamCurr;
				bSaveHMISvyConfig := FALSE;  //new for Hermes 1.3

				tyCommon.tySet.tyBtnSave.bRtCompl 	:= FALSE;
				fUIInRtStatOff(ADR(tyCommon.tySet.tyBtnSave.uiMaskRtStat));

			END_IF

		END_IF

	END_IF

END_ACTION
```

#### Act_OptP1022Keypad.st
```iecst
ACTION Act_OptP1022Keypad:

	IF fUIOutRtStatTPIsOpen(ADR(tyP1022McSetVComm.tyVComSvy.tyNumSndAliveTm.uiRtStat)) = TRUE THEN
		tyProperty.tyKeypad.tyTxtTitle.sTxt	:= tyP1022McSetVComm.tyVComSvy.tyNumSndAliveTm.sKeypadTitle;

	ELSIF fUIOutRtStatTPIsOpen(ADR(tyP1022McSetVComm.tyVComSvy.tyNumSvySystemPort.uiRtStat)) = TRUE THEN
		tyProperty.tyKeypad.tyTxtTitle.sTxt	:= tyP1022McSetVComm.tyVComSvy.tyNumSvySystemPort.sKeypadTitle;

	END_IF

END_ACTION
```

#### Act_EntP1023Disp.st
```iecst
ACTION Act_EntP1023Disp:

	//Access Address
	IF p_tyNtParamCurr.bProjLaneBPrep THEN
		p_tyC0004Navi ACCESS ADR(tyP1023McSetHComm.tyNaviLyr1);
	ELSE
		p_tyC0004Navi ACCESS ADR(tyP1023McSetHComm.tyNaviBack);
	END_IF

	p_tyC0005Main ACCESS ADR(tyCommon.tyMain);

	p_tyC0006Set ACCESS ADR(tyCommon.tySet);

	p_tyC0007Notif ACCESS ADR(tyCommon.tyNotif);

	p_tyC0008MsgBox ACCESS ADR(tyP1023McSetHComm.tyMsgBoxHide);

	p_tyC0009Info ACCESS ADR(tyCommon.tyInfo);

	p_tyP1023McSetHCommUSSel ACCESS ADR(tyP1023McSetHComm.tyUSSelA);
	p_tyP1023McSetHCommUSSMEMA ACCESS ADR(tyP1023McSetHComm.tyUSSMEMAA);
	p_tyP1023McSetHCommUSHermes ACCESS ADR(tyP1023McSetHComm.tyUSHermesA);

	//Backup Param
	tyP1023McSetHComm.tyUSSelABkUp		:= tyP1023McSetHComm.tyUSSelA;
	tyP1023McSetHComm.tyUSSMEMAABkUp	:= tyP1023McSetHComm.tyUSSMEMAA;
	tyP1023McSetHComm.tyUSHermesABkUp	:= tyP1023McSetHComm.tyUSHermesA;
	tyP1023McSetHComm.tyUSSelBBkUp		:= tyP1023McSetHComm.tyUSSelB;
	tyP1023McSetHComm.tyUSSMEMABBkUp	:= tyP1023McSetHComm.tyUSSMEMAB;
	tyP1023McSetHComm.tyUSHermesBBkUp	:= tyP1023McSetHComm.tyUSHermesB;

END_ACTION
```

#### Act_ExitP1023.st
```iecst
ACTION Act_ExitP1023:

	IF tyCommon.tySet.tyBtnSave.uiMaskRtStat.0 = FALSE THEN
		usiChgPage	:= 1;

	ELSE

		p_tyC0008MsgBox ACCESS ADR(tyP1023McSetHComm.tyMsgBoxExitAsk);

		IF tyP1023McSetHComm.tyMsgBoxExitAsk.tyBtnYes.bRtCompl = TRUE THEN
			tyP1023McSetHComm.tyMsgBoxExitAsk.tyBtnYes.bRtCompl	:= FALSE;
			tyP1023McSetHComm.tyMsgBoxExitAsk.tyBtnYes.bValue	:= FALSE;

			p_tyC0008MsgBox ACCESS ADR(tyP1023McSetHComm.tyMsgBoxHide);

			//Restore Param
			tyP1023McSetHComm.tyUSSelA		:= tyP1023McSetHComm.tyUSSelABkUp;
			tyP1023McSetHComm.tyUSSMEMAA	:= tyP1023McSetHComm.tyUSSMEMAABkUp;
			tyP1023McSetHComm.tyUSHermesA	:= tyP1023McSetHComm.tyUSHermesABkUp;

			tyP1023McSetHComm.tyUSSelB		:= tyP1023McSetHComm.tyUSSelBBkUp;
			tyP1023McSetHComm.tyUSSMEMAB	:= tyP1023McSetHComm.tyUSSMEMABBkUp;
			tyP1023McSetHComm.tyUSHermesB	:= tyP1023McSetHComm.tyUSHermesBBkUp;

			fUIInRtStatOff(ADR(tyCommon.tySet.tyBtnSave.uiMaskRtStat));

			usiChgPage	:= 1;

		ELSIF tyP1023McSetHComm.tyMsgBoxExitAsk.tyBtnNo.bRtCompl = TRUE THEN
			tyP1023McSetHComm.tyMsgBoxExitAsk.tyBtnNo.bRtCompl	:= FALSE;
			tyP1023McSetHComm.tyMsgBoxExitAsk.tyBtnNo.bValue	:= FALSE;

			p_tyC0008MsgBox ACCESS ADR(tyP1023McSetHComm.tyMsgBoxHide);

			eChgPage	:= eCurrPage;
			usiChgPage	:= 0;

		END_IF

	END_IF

END_ACTION
```

#### Act_OptP1023Navi.st
```iecst
ACTION Act_OptP1023Navi:

	tyP1023McSetHComm.tyNaviBack.tyBtnBack.bRtLk	:= tyCommon.tySet.tyBtnSave.bRtCompl;
	tyP1023McSetHComm.tyNaviLyr1.tyBtnBack.bRtLk	:= tyCommon.tySet.tyBtnSave.bRtCompl;
	tyP1023McSetHComm.tyNaviLyr2.tyBtnBack.bRtLk	:= tyCommon.tySet.tyBtnSave.bRtCompl;

	IF tyP1023McSetHComm.tyNaviLyr1.tyBtnBack.bRtCompl = TRUE OR tyP1023McSetHComm.tyNaviLyr2.tyBtnBack.bRtCompl = TRUE OR tyP1023McSetHComm.tyNaviBack.tyBtnBack.bRtCompl = TRUE THEN
		eChgPage	:= UIP1020McSetNavi;

		tyP1023McSetHComm.tyNaviLyr1.tyBtnBack.bRtCompl		:= FALSE;
		tyP1023McSetHComm.tyNaviLyr2.tyBtnBack.bRtCompl		:= FALSE;
		tyP1023McSetHComm.tyNaviBack.tyBtnBack.bRtCompl		:= FALSE;

	ELSIF tyP1023McSetHComm.tyNaviLyr1.tyBtnLeft.bRtCompl = TRUE OR tyP1023McSetHComm.tyNaviLyr1.tyBtnRgt.bRtCompl = TRUE THEN

		p_tyC0004Navi ACCESS ADR(tyP1023McSetHComm.tyNaviLyr2);
		p_tyP1023McSetHCommUSSel ACCESS ADR(tyP1023McSetHComm.tyUSSelB);
		p_tyP1023McSetHCommUSSMEMA ACCESS ADR(tyP1023McSetHComm.tyUSSMEMAB);
		p_tyP1023McSetHCommUSHermes ACCESS ADR(tyP1023McSetHComm.tyUSHermesB);

		tyP1023McSetHComm.tyUSSelB.tyBtnHermes.uiRtStat.0	:= NOT p_tyNtParamCurr.bHermesPrep;

		tyP1023McSetHComm.tyNaviLyr1.tyBtnLeft.bRtCompl	:= FALSE;
		tyP1023McSetHComm.tyNaviLyr1.tyBtnRgt.bRtCompl	:= FALSE;

	ELSIF tyP1023McSetHComm.tyNaviLyr2.tyBtnLeft.bRtCompl = TRUE OR tyP1023McSetHComm.tyNaviLyr2.tyBtnRgt.bRtCompl = TRUE THEN

		p_tyC0004Navi ACCESS ADR(tyP1023McSetHComm.tyNaviLyr1);
		p_tyP1023McSetHCommUSSel ACCESS ADR(tyP1023McSetHComm.tyUSSelA);
		p_tyP1023McSetHCommUSSMEMA ACCESS ADR(tyP1023McSetHComm.tyUSSMEMAA);
		p_tyP1023McSetHCommUSHermes ACCESS ADR(tyP1023McSetHComm.tyUSHermesA);

		tyP1023McSetHComm.tyUSSelA.tyBtnHermes.uiRtStat.0	:= NOT p_tyNtParamCurr.bHermesPrep;

		tyP1023McSetHComm.tyNaviLyr2.tyBtnLeft.bRtCompl	:= FALSE;
		tyP1023McSetHComm.tyNaviLyr2.tyBtnRgt.bRtCompl	:= FALSE;

	END_IF

END_ACTION
```

#### Act_OptP1023ShowLyr.st
```iecst
ACTION Act_OptP1023ShowLyr:

	//Upstream A
	IF tyP1023McSetHComm.tyUSSelA.tyLyr.uiRtStat.0 = FALSE THEN

		IF tyP1023McSetHComm.tyUSSelA.tyBtnSMEMA.bValue = TRUE THEN

			fUIInRtStatOff(ADR(tyP1023McSetHComm.tyUSSMEMAA.tyLyr.uiRtStat));
			fUIInRtStatHide(ADR(tyP1023McSetHComm.tyUSHermesA.tyLyr.uiRtStat));

			tyP1023McSetHComm.tyUSSMEMAA.tyBtnGdSig.uiRtStat.0	:= NOT(tyP1023McSetHComm.tyUSSMEMAA.tyDrpDnSMEMAMod.usiValueIdx = 2);

		ELSIF tyP1023McSetHComm.tyUSSelA.tyBtnHermes.bValue = TRUE THEN

			fUIInRtStatHide(ADR(tyP1023McSetHComm.tyUSSMEMAA.tyLyr.uiRtStat));
			fUIInRtStatOff(ADR(tyP1023McSetHComm.tyUSHermesA.tyLyr.uiRtStat));

			//Mask
			tyP1023McSetHComm.tyUSHermesA.tyBitmapMask.uiRtStat.0	:= NOT(p_tyNtParamCurr.bHermesRmtPrep = TRUE AND p_tyMcParamCurr.bHermesRmtEn = TRUE);
		END_IF

	ELSE

		fUIInRtStatHide(ADR(tyP1023McSetHComm.tyUSSMEMAA.tyLyr.uiRtStat));
		fUIInRtStatHide(ADR(tyP1023McSetHComm.tyUSHermesA.tyLyr.uiRtStat));

	END_IF

	//Upstream B
	IF tyP1023McSetHComm.tyUSSelB.tyLyr.uiRtStat.0 = FALSE THEN

		IF tyP1023McSetHComm.tyUSSelB.tyBtnSMEMA.bValue = TRUE THEN

			fUIInRtStatOff(ADR(tyP1023McSetHComm.tyUSSMEMAB.tyLyr.uiRtStat));
			fUIInRtStatHide(ADR(tyP1023McSetHComm.tyUSHermesB.tyLyr.uiRtStat));

			tyP1023McSetHComm.tyUSSMEMAB.tyBtnGdSig.uiRtStat.0	:= NOT(tyP1023McSetHComm.tyUSSMEMAB.tyDrpDnSMEMAMod.usiValueIdx = 2);

		ELSIF tyP1023McSetHComm.tyUSSelB.tyBtnHermes.bValue = TRUE THEN

			fUIInRtStatHide(ADR(tyP1023McSetHComm.tyUSSMEMAB.tyLyr.uiRtStat));
			fUIInRtStatOff(ADR(tyP1023McSetHComm.tyUSHermesB.tyLyr.uiRtStat));

			//Mask
			tyP1023McSetHComm.tyUSHermesB.tyBitmapMask.uiRtStat.0	:= NOT(p_tyNtParamCurr.bHermesRmtPrep = TRUE AND p_tyMcParamCurr.bHermesRmtEn = TRUE);
		END_IF

	ELSE

		fUIInRtStatHide(ADR(tyP1023McSetHComm.tyUSSMEMAB.tyLyr.uiRtStat));
		fUIInRtStatHide(ADR(tyP1023McSetHComm.tyUSHermesB.tyLyr.uiRtStat));

	END_IF

END_ACTION
```

#### Act_OptP1023USSel.st
```iecst
ACTION Act_OptP1023USSel:

	//Select SMEMA Communication A
	IF tyP1023McSetHComm.tyUSSelA.tyBtnSMEMA.bRtCompl = TRUE THEN
		tyP1023McSetHComm.tyUSSelA.tyBtnSMEMA.bRtCompl	:= FALSE;

		tyP1023McSetHComm.tyUSSelA.tyBtnSMEMA.bValue	:= TRUE;
		tyP1023McSetHComm.tyUSSelA.tyBtnSMEMA.bRtLk		:= TRUE;

		tyP1023McSetHComm.tyUSSelA.tyBtnHermes.bValue	:= FALSE;
		tyP1023McSetHComm.tyUSSelA.tyBtnHermes.bRtLk	:= FALSE;

	//Select Hermes Communication A
	ELSIF tyP1023McSetHComm.tyUSSelA.tyBtnHermes.bRtCompl = TRUE THEN
		tyP1023McSetHComm.tyUSSelA.tyBtnHermes.bRtCompl	:= FALSE;

		tyP1023McSetHComm.tyUSSelA.tyBtnSMEMA.bValue	:= FALSE;
		tyP1023McSetHComm.tyUSSelA.tyBtnSMEMA.bRtLk		:= FALSE;

		tyP1023McSetHComm.tyUSSelA.tyBtnHermes.bValue	:= TRUE;
		tyP1023McSetHComm.tyUSSelA.tyBtnHermes.bRtLk	:= TRUE;

	END_IF

	//Select SMEMA Communication B
	IF tyP1023McSetHComm.tyUSSelB.tyBtnSMEMA.bRtCompl = TRUE THEN
		tyP1023McSetHComm.tyUSSelB.tyBtnSMEMA.bRtCompl	:= FALSE;

		tyP1023McSetHComm.tyUSSelB.tyBtnSMEMA.bValue	:= TRUE;
		tyP1023McSetHComm.tyUSSelB.tyBtnSMEMA.bRtLk		:= TRUE;

		tyP1023McSetHComm.tyUSSelB.tyBtnHermes.bValue	:= FALSE;
		tyP1023McSetHComm.tyUSSelB.tyBtnHermes.bRtLk	:= FALSE;

		//Select Hermes Communication B
	ELSIF tyP1023McSetHComm.tyUSSelB.tyBtnHermes.bRtCompl = TRUE THEN
		tyP1023McSetHComm.tyUSSelB.tyBtnHermes.bRtCompl	:= FALSE;

		tyP1023McSetHComm.tyUSSelB.tyBtnSMEMA.bValue	:= FALSE;
		tyP1023McSetHComm.tyUSSelB.tyBtnSMEMA.bRtLk		:= FALSE;

		tyP1023McSetHComm.tyUSSelB.tyBtnHermes.bValue	:= TRUE;
		tyP1023McSetHComm.tyUSSelB.tyBtnHermes.bRtLk	:= TRUE;

	END_IF

END_ACTION
```

#### Act_OptP1023Save.st
```iecst
ACTION Act_OptP1023Save:

	IF tyP1023McSetHComm.tyUSSelA.tyBtnSMEMA.bRtCompl						OR tyP1023McSetHComm.tyUSSelA.tyBtnHermes.bRtCompl
		OR tyP1023McSetHComm.tyUSSMEMAA.tyDrpDnSMEMAMod.bRtCompl			OR tyP1023McSetHComm.tyUSSMEMAA.tyBtnGdSig.bRtCompl
		OR tyP1023McSetHComm.tyUSHermesA.tyNumSndAliveTm.bRtCompl 			OR tyP1023McSetHComm.tyUSHermesA.tyNumLaneID.bRtCompl
		OR tyP1023McSetHComm.tyUSHermesA.tyStringHostAddr.bRtCompl			OR tyP1023McSetHComm.tyUSHermesA.tyNumHostPort.bRtCompl
		OR tyP1023McSetHComm.tyUSHermesA.tyBtnCheckAliveResponse.bRtCompl 	OR tyP1023McSetHComm.tyUSHermesA.tyBtnCmpParam.bRtCompl
		OR tyP1023McSetHComm.tyUSHermesA.tyBtnCmpTypeId.bRtCompl			OR tyP1023McSetHComm.tyUSHermesA.tyBtnOverWrite.bRtCompl
		OR tyP1023McSetHComm.tyUSHermesA.tyBtnBoardForecast.bRtCompl		OR tyP1023McSetHComm.tyUSHermesA.tyBtnQueryBoardInfo.bRtCompl

		OR tyP1023McSetHComm.tyUSSelB.tyBtnSMEMA.bRtCompl					OR tyP1023McSetHComm.tyUSSelB.tyBtnHermes.bRtCompl
		OR tyP1023McSetHComm.tyUSSMEMAB.tyDrpDnSMEMAMod.bRtCompl			OR tyP1023McSetHComm.tyUSSMEMAB.tyBtnGdSig.bRtCompl
		OR tyP1023McSetHComm.tyUSHermesB.tyNumSndAliveTm.bRtCompl 			OR tyP1023McSetHComm.tyUSHermesB.tyNumLaneID.bRtCompl
		OR tyP1023McSetHComm.tyUSHermesB.tyStringHostAddr.bRtCompl			OR tyP1023McSetHComm.tyUSHermesB.tyNumHostPort.bRtCompl
		OR tyP1023McSetHComm.tyUSHermesB.tyBtnCheckAliveResponse.bRtCompl	OR tyP1023McSetHComm.tyUSHermesB.tyBtnCmpParam.bRtCompl
		OR tyP1023McSetHComm.tyUSHermesB.tyBtnCmpTypeId.bRtCompl			OR tyP1023McSetHComm.tyUSHermesB.tyBtnOverWrite.bRtCompl
		OR tyP1023McSetHComm.tyUSHermesB.tyBtnBoardForecast.bRtCompl			OR tyP1023McSetHComm.tyUSHermesB.tyBtnQueryBoardInfo.bRtCompl THEN
		fUIInRtStatHide(ADR(tyCommon.tySet.tyBtnSave.uiMaskRtStat));

		tyP1023McSetHComm.tyUSSMEMAA.tyDrpDnSMEMAMod.bRtCompl				:= FALSE;
		tyP1023McSetHComm.tyUSSMEMAA.tyBtnGdSig.bRtCompl					:= FALSE;
		tyP1023McSetHComm.tyUSHermesA.tyNumSndAliveTm.bRtCompl				:= FALSE;
		tyP1023McSetHComm.tyUSHermesA.tyNumLaneID.bRtCompl					:= FALSE;
		tyP1023McSetHComm.tyUSHermesA.tyStringHostAddr.bRtCompl				:= FALSE;
		tyP1023McSetHComm.tyUSHermesA.tyNumHostPort.bRtCompl				:= FALSE;
		tyP1023McSetHComm.tyUSHermesA.tyBtnCheckAliveResponse.bRtCompl		:= FALSE;
		tyP1023McSetHComm.tyUSHermesA.tyBtnCmpParam.bRtCompl				:= FALSE;
		tyP1023McSetHComm.tyUSHermesA.tyBtnCmpTypeId.bRtCompl				:= FALSE;
		tyP1023McSetHComm.tyUSHermesA.tyBtnOverWrite.bRtCompl				:= FALSE;
		tyP1023McSetHComm.tyUSHermesA.tyBtnBoardForecast.bRtCompl			:= FALSE;
		tyP1023McSetHComm.tyUSHermesA.tyBtnQueryBoardInfo.bRtCompl			:= FALSE;

		tyP1023McSetHComm.tyUSSMEMAB.tyDrpDnSMEMAMod.bRtCompl				:= FALSE;
		tyP1023McSetHComm.tyUSSMEMAB.tyBtnGdSig.bRtCompl					:= FALSE;
		tyP1023McSetHComm.tyUSHermesB.tyNumSndAliveTm.bRtCompl				:= FALSE;
		tyP1023McSetHComm.tyUSHermesB.tyNumLaneID.bRtCompl					:= FALSE;
		tyP1023McSetHComm.tyUSHermesB.tyStringHostAddr.bRtCompl				:= FALSE;
		tyP1023McSetHComm.tyUSHermesB.tyNumHostPort.bRtCompl				:= FALSE;
		tyP1023McSetHComm.tyUSHermesB.tyBtnCheckAliveResponse.bRtCompl		:= FALSE;
		tyP1023McSetHComm.tyUSHermesB.tyBtnCmpParam.bRtCompl				:= FALSE;
		tyP1023McSetHComm.tyUSHermesB.tyBtnCmpTypeId.bRtCompl				:= FALSE;
		tyP1023McSetHComm.tyUSHermesB.tyBtnOverWrite.bRtCompl				:= FALSE;
		tyP1023McSetHComm.tyUSHermesB.tyBtnBoardForecast.bRtCompl			:= FALSE;
		tyP1023McSetHComm.tyUSHermesB.tyBtnQueryBoardInfo.bRtCompl			:= FALSE;
	END_IF

	//new for Hermes 1.3
	//Auto de-select
	IF EDGEPOS(tyP1023McSetHComm.tyUSHermesA.tyBtnCmpTypeId.bValue) THEN
		tyP1023McSetHComm.tyUSHermesA.tyBtnOverWrite.bValue := FALSE;
	ELSIF EDGEPOS(tyP1023McSetHComm.tyUSHermesA.tyBtnCmpParam.bValue) THEN
		tyP1023McSetHComm.tyUSHermesA.tyBtnCmpTypeId.bValue := TRUE;
	ELSIF EDGEPOS(tyP1023McSetHComm.tyUSHermesA.tyBtnCmpTypeId.bValue = FALSE) THEN
		tyP1023McSetHComm.tyUSHermesA.tyBtnCmpParam.bValue := FALSE;
	ELSIF EDGEPOS(tyP1023McSetHComm.tyUSHermesA.tyBtnOverWrite.bValue = TRUE) THEN
		tyP1023McSetHComm.tyUSHermesA.tyBtnCmpTypeId.bValue := FALSE;
	END_IF

	IF EDGEPOS(tyP1023McSetHComm.tyUSHermesB.tyBtnCmpTypeId.bValue) THEN
		tyP1023McSetHComm.tyUSHermesB.tyBtnOverWrite.bValue := FALSE;
	ELSIF EDGEPOS(tyP1023McSetHComm.tyUSHermesB.tyBtnCmpParam.bValue) THEN
		tyP1023McSetHComm.tyUSHermesB.tyBtnCmpTypeId.bValue := TRUE;
	ELSIF EDGEPOS(tyP1023McSetHComm.tyUSHermesB.tyBtnCmpTypeId.bValue = FALSE) THEN
		tyP1023McSetHComm.tyUSHermesB.tyBtnCmpParam.bValue := FALSE;
	ELSIF EDGEPOS(tyP1023McSetHComm.tyUSHermesB.tyBtnOverWrite.bValue = TRUE) THEN
		tyP1023McSetHComm.tyUSHermesB.tyBtnCmpTypeId.bValue := FALSE;
	END_IF

	IF tyCommon.tySet.tyBtnSave.bRtCompl = TRUE THEN

		IF usiSaveCommStep = 0 THEN
			//Verify Hermes A IP Address
			IF (tyP1023McSetHComm.tyUSSelA.tyBtnHermes.bValue = TRUE) AND NOT(p_tyNtParamCurr.bHermesRmtPrep = TRUE AND p_tyMcParamCurr.bHermesRmtEn = TRUE) THEN
				IF fIPValid(tyP1023McSetHComm.tyUSHermesA.tyStringHostAddr.sValue, ADR(a_iIPPart1)) = TRUE THEN
					usiSaveCommStep	:= 1;
				ELSE
					usiSaveCommStep	:= 99;
				END_IF
			ELSE
				usiSaveCommStep	:= 1;
			END_IF

		ELSIF usiSaveCommStep = 1 THEN
			//Verify Hermes B IP Address
			IF (p_tyNtParamCurr.bProjLaneBPrep = TRUE) AND (tyP1023McSetHComm.tyUSSelB.tyBtnHermes.bValue = TRUE) AND NOT(p_tyNtParamCurr.bHermesRmtPrep = TRUE AND p_tyMcParamCurr.bHermesRmtEn = TRUE) THEN
				IF fIPValid(tyP1023McSetHComm.tyUSHermesB.tyStringHostAddr.sValue, ADR(a_iIPPart1)) = TRUE THEN
					usiSaveCommStep	:= 2;
				ELSE
					usiSaveCommStep	:= 99;
				END_IF
			ELSE
				usiSaveCommStep	:= 2;
			END_IF

		ELSIF usiSaveCommStep = 2 THEN
			//Save Machine Parameter
			//Upstream A
			IF tyP1023McSetHComm.tyUSSelA.tyBtnSMEMA.bValue = TRUE THEN
				tyMcParamWr.eUSCommA	:= McSetCommModSMEMA;
			ELSIF tyP1023McSetHComm.tyUSSelA.tyBtnHermes.bValue = TRUE THEN
				tyMcParamWr.eUSCommA	:= McSetCommModHermes;
			END_IF

			tyMcParamWr.tyUSCommASMEMA.eSelection		:= USINT_TO_UDINT(tyP1023McSetHComm.tyUSSMEMAA.tyDrpDnSMEMAMod.usiValueIdx);
			tyMcParamWr.tyUSCommASMEMA.bStatSigSetGd	:= tyP1023McSetHComm.tyUSSMEMAA.tyBtnGdSig.bValue;

			//Upstream B
			IF tyP1023McSetHComm.tyUSSelB.tyBtnSMEMA.bValue = TRUE THEN
				tyMcParamWr.eUSCommB	:= McSetCommModSMEMA;
			ELSIF tyP1023McSetHComm.tyUSSelB.tyBtnHermes.bValue = TRUE THEN
				tyMcParamWr.eUSCommB	:= McSetCommModHermes;
			END_IF

			tyMcParamWr.tyUSCommBSMEMA.eSelection		:= USINT_TO_UDINT(tyP1023McSetHComm.tyUSSMEMAB.tyDrpDnSMEMAMod.usiValueIdx);
			tyMcParamWr.tyUSCommBSMEMA.bStatSigSetGd	:= tyP1023McSetHComm.tyUSSMEMAB.tyBtnGdSig.bValue;

			eMcParamAct	:= McParamActWrite;

			IF p_eMcParamStat = McParamActWrite AND p_eMcParamStatus = Done THEN
				eMcParamAct	:= McParamActIdle;

				//Update BackUp Param
				tyP1023McSetHComm.tyUSSelABkUp 		:= tyP1023McSetHComm.tyUSSelA;
				tyP1023McSetHComm.tyUSSMEMAABkUp	:= tyP1023McSetHComm.tyUSSMEMAA;
				tyP1023McSetHComm.tyUSSelBBkUp		:= tyP1023McSetHComm.tyUSSelB;
				tyP1023McSetHComm.tyUSSMEMABBkUp	:= tyP1023McSetHComm.tyUSSMEMAB;

				usiSaveCommStep	:= 3;

			ELSIF p_eMcParamStatus = Error THEN
				p_tyC0008MsgBox ACCESS ADR(tyP1023McSetHComm.tyMsgBoxSaveErr);

				IF tyP1023McSetHComm.tyMsgBoxSaveErr.tyBtnNo.bRtCompl = TRUE THEN
					tyP1023McSetHComm.tyMsgBoxSaveErr.tyBtnNo.bRtCompl	:= FALSE;
					tyP1023McSetHComm.tyMsgBoxSaveErr.tyBtnNo.bValue	:= FALSE;

					p_tyC0008MsgBox ACCESS ADR(tyP1023McSetHComm.tyMsgBoxHide);

					//Restore Param
					tyP1023McSetHComm.tyUSSelA		:= tyP1023McSetHComm.tyUSSelABkUp;
					tyP1023McSetHComm.tyUSSMEMAA	:= tyP1023McSetHComm.tyUSSMEMAABkUp;
					tyP1023McSetHComm.tyUSSelB		:= tyP1023McSetHComm.tyUSSelBBkUp;
					tyP1023McSetHComm.tyUSSMEMAB	:= tyP1023McSetHComm.tyUSSMEMABBkUp;

					tyMcParamWr	:= p_tyMcParamCurr;

					usiSaveCommStep	:= 3;
				END_IF

			END_IF

		ELSIF usiSaveCommStep = 3 THEN
			//Save Hermes Configuration
			//Upstream A
			a_tyHermesUSParamWr[0].tSndAlive					:= DINT_TO_TIME(tyP1023McSetHComm.tyUSHermesA.tyNumSndAliveTm.diValue);
			a_tyHermesUSParamWr[0].iLaneID						:= DINT_TO_INT(tyP1023McSetHComm.tyUSHermesA.tyNumLaneID.diValue);
			a_tyHermesUSParamWr[0].sHostAddress					:= tyP1023McSetHComm.tyUSHermesA.tyStringHostAddr.sValue;
			a_tyHermesUSParamWr[0].uiHostPort					:= DINT_TO_UINT(tyP1023McSetHComm.tyUSHermesA.tyNumHostPort.diValue);
			a_tyHermesUSParamWr[0].bFeatureCheckAliveResponse	:= tyP1023McSetHComm.tyUSHermesA.tyBtnCheckAliveResponse.bValue;
			a_tyHermesUSParamWr[0].bCmpTypeId					:= tyP1023McSetHComm.tyUSHermesA.tyBtnCmpTypeId.bValue;
			a_tyHermesUSParamWr[0].bCmpParam					:= tyP1023McSetHComm.tyUSHermesA.tyBtnCmpParam.bValue;
			a_tyHermesUSParamWr[0].bOverwrite					:= tyP1023McSetHComm.tyUSHermesA.tyBtnOverWrite.bValue;
			a_tyHermesUSParamWr[0].bFeatureBoardForecast		:= tyP1023McSetHComm.tyUSHermesA.tyBtnBoardForecast.bValue;
			a_tyHermesUSParamWr[0].bFeatureQueryBoardInfo		:= tyP1023McSetHComm.tyUSHermesA.tyBtnQueryBoardInfo.bValue;
			//Upstream B
			a_tyHermesUSParamWr[1].tSndAlive					:= DINT_TO_TIME(tyP1023McSetHComm.tyUSHermesB.tyNumSndAliveTm.diValue);
			a_tyHermesUSParamWr[1].iLaneID						:= DINT_TO_INT(tyP1023McSetHComm.tyUSHermesB.tyNumLaneID.diValue);
			a_tyHermesUSParamWr[1].sHostAddress					:= tyP1023McSetHComm.tyUSHermesB.tyStringHostAddr.sValue;
			a_tyHermesUSParamWr[1].uiHostPort					:= DINT_TO_UINT(tyP1023McSetHComm.tyUSHermesB.tyNumHostPort.diValue);
			a_tyHermesUSParamWr[1].bFeatureCheckAliveResponse	:= tyP1023McSetHComm.tyUSHermesB.tyBtnCheckAliveResponse.bValue;
			a_tyHermesUSParamWr[1].bCmpTypeId					:= tyP1023McSetHComm.tyUSHermesB.tyBtnCmpTypeId.bValue;
			a_tyHermesUSParamWr[1].bCmpParam					:= tyP1023McSetHComm.tyUSHermesB.tyBtnCmpParam.bValue;
			a_tyHermesUSParamWr[1].bOverwrite					:= tyP1023McSetHComm.tyUSHermesB.tyBtnOverWrite.bValue;
			a_tyHermesUSParamWr[1].bFeatureBoardForecast		:= tyP1023McSetHComm.tyUSHermesB.tyBtnBoardForecast.bValue;
			a_tyHermesUSParamWr[1].bFeatureQueryBoardInfo		:= tyP1023McSetHComm.tyUSHermesB.tyBtnQueryBoardInfo.bValue;

			bSaveHMIConfigure := TRUE;

			eHermesAct	:= HermesActWriteConfig;

			IF p_eHermesStat = HermesActWriteConfig AND p_eHermesStatus = Done THEN
				eHermesAct	:= HermesActIdle;

				//Update BackUp Param
				tyP1023McSetHComm.tyUSHermesABkUp	:= tyP1023McSetHComm.tyUSHermesA;
				tyP1023McSetHComm.tyUSHermesBBkUp	:= tyP1023McSetHComm.tyUSHermesB;

				usiSaveCommStep	:= 0;
				bSaveHMIConfigure := FALSE;

				tyCommon.tySet.tyBtnSave.bRtCompl	:= FALSE;

				fUIInRtStatOff(ADR(tyCommon.tySet.tyBtnSave.uiMaskRtStat));

			ELSIF p_eMcParamStatus = Error THEN
				p_tyC0008MsgBox ACCESS ADR(tyP1023McSetHComm.tyMsgBoxSaveErr);

				IF tyP1023McSetHComm.tyMsgBoxSaveErr.tyBtnNo.bRtCompl = TRUE THEN
					tyP1023McSetHComm.tyMsgBoxSaveErr.tyBtnNo.bRtCompl	:= FALSE;
					tyP1023McSetHComm.tyMsgBoxSaveErr.tyBtnNo.bValue	:= FALSE;

					p_tyC0008MsgBox ACCESS ADR(tyP1023McSetHComm.tyMsgBoxHide);

					//Restore Param
					tyP1023McSetHComm.tyUSHermesA	:= tyP1023McSetHComm.tyUSHermesABkUp;
					tyP1023McSetHComm.tyUSHermesB	:= tyP1023McSetHComm.tyUSHermesBBkUp;

					a_tyHermesUSParamWr				:= p_tyHermesConfiguration.a_tyUSParam;

					tyCommon.tySet.tyBtnSave.bRtCompl	:= FALSE;
					bSaveHMIConfigure := FALSE;
					fUIInRtStatOff(ADR(tyCommon.tySet.tyBtnSave.uiMaskRtStat));
					usiSaveCommStep	:= 0;
				END_IF

			END_IF

		ELSIF usiSaveCommStep = 99 THEN
			//Message: IP Address Invalid
			p_tyC0008MsgBox ACCESS ADR(tyP1023McSetHComm.tyMsgBoxIPAddrInvalid);

			IF tyP1023McSetHComm.tyMsgBoxIPAddrInvalid.tyBtnNo.bRtCompl = TRUE THEN
				tyP1023McSetHComm.tyMsgBoxIPAddrInvalid.tyBtnNo.bRtCompl	:= FALSE;
				tyP1023McSetHComm.tyMsgBoxIPAddrInvalid.tyBtnNo.bValue		:= FALSE;

				p_tyC0008MsgBox ACCESS ADR(tyP1023McSetHComm.tyMsgBoxHide);

				//Restore Param
				tyP1023McSetHComm.tyUSSelA		:= tyP1023McSetHComm.tyUSSelABkUp;
				tyP1023McSetHComm.tyUSSMEMAA	:= tyP1023McSetHComm.tyUSSMEMAABkUp;
				tyP1023McSetHComm.tyUSHermesA	:= tyP1023McSetHComm.tyUSHermesABkUp;
				tyP1023McSetHComm.tyUSSelB		:= tyP1023McSetHComm.tyUSSelBBkUp;
				tyP1023McSetHComm.tyUSSMEMAB	:= tyP1023McSetHComm.tyUSSMEMABBkUp;
				tyP1023McSetHComm.tyUSHermesB	:= tyP1023McSetHComm.tyUSHermesBBkUp;

				tyCommon.tySet.tyBtnSave.bRtCompl	:= FALSE;

				fUIInRtStatOff(ADR(tyCommon.tySet.tyBtnSave.uiMaskRtStat));

				usiSaveCommStep	:= 0;
			END_IF

		END_IF

	END_IF

	//Added Siemen
	IF  p_tyNtParamCurr.eCustomerReq = Siemens AND
		tyMcParamWr.eUSCommA <> p_tyMcParamCurr.eUSCommA
		AND usiSaveCommStep = 2
		AND tyCommon.tySet.tyBtnSave.bRtCompl	= TRUE THEN
			usiHComModChaged := usiHComModChaged + 1;
	END_IF
END_ACTION
```

#### Act_OptP1023Keypad.st
```iecst
ACTION Act_OptP1023Keypad:

	//Upstream A
	IF fUIOutRtStatTPIsOpen(ADR(tyP1023McSetHComm.tyUSHermesA.tyNumSndAliveTm.uiRtStat)) = TRUE THEN
		tyProperty.tyKeypad.tyStringTitle.sKeypadTitle	:= tyP1023McSetHComm.tyUSHermesA.tyNumSndAliveTm.sKeypadTitle;

	ELSIF fUIOutRtStatTPIsOpen(ADR(tyP1023McSetHComm.tyUSHermesA.tyNumLaneID.uiRtStat)) = TRUE THEN
		tyProperty.tyKeypad.tyStringTitle.sKeypadTitle	:= tyP1023McSetHComm.tyUSHermesA.tyNumLaneID.sKeypadTitle;

	ELSIF fUIOutRtStatTPIsOpen(ADR(tyP1023McSetHComm.tyUSHermesA.tyNumHostPort.uiRtStat)) = TRUE THEN
		tyProperty.tyKeypad.tyStringTitle.sKeypadTitle	:= tyP1023McSetHComm.tyUSHermesA.tyNumHostPort.sKeypadTitle;

	ELSIF fUIOutRtStatTPIsOpen(ADR(tyP1023McSetHComm.tyUSHermesA.tyStringHostAddr.uiRtStat)) = TRUE THEN
		tyProperty.tyKeypad.tyStringTitle.sKeypadTitle	:= tyP1023McSetHComm.tyUSHermesA.tyStringHostAddr.sKeypadTitle;

	END_IF

	//Upstream B
	IF fUIOutRtStatTPIsOpen(ADR(tyP1023McSetHComm.tyUSHermesB.tyNumSndAliveTm.uiRtStat)) = TRUE THEN
		tyProperty.tyKeypad.tyStringTitle.sKeypadTitle	:= tyP1023McSetHComm.tyUSHermesB.tyNumSndAliveTm.sKeypadTitle;

	ELSIF fUIOutRtStatTPIsOpen(ADR(tyP1023McSetHComm.tyUSHermesB.tyNumLaneID.uiRtStat)) = TRUE THEN
		tyProperty.tyKeypad.tyStringTitle.sKeypadTitle	:= tyP1023McSetHComm.tyUSHermesB.tyNumLaneID.sKeypadTitle;

	ELSIF fUIOutRtStatTPIsOpen(ADR(tyP1023McSetHComm.tyUSHermesB.tyNumHostPort.uiRtStat)) = TRUE THEN
		tyProperty.tyKeypad.tyStringTitle.sKeypadTitle	:= tyP1023McSetHComm.tyUSHermesB.tyNumHostPort.sKeypadTitle;

	ELSIF fUIOutRtStatTPIsOpen(ADR(tyP1023McSetHComm.tyUSHermesB.tyStringHostAddr.uiRtStat)) = TRUE THEN
		tyProperty.tyKeypad.tyStringTitle.sKeypadTitle	:= tyP1023McSetHComm.tyUSHermesB.tyStringHostAddr.sKeypadTitle;

	END_IF

END_ACTION
```

#### Act_EntP1024Disp.st
```iecst
ACTION Act_EntP1024Disp:

	//Access Address
	p_tyC0004Navi ACCESS ADR(tyP1024McSetAntiGap.tyNaviBack);

	p_tyC0005Main ACCESS ADR(tyCommon.tyMain);

	p_tyC0006Set ACCESS ADR(tyCommon.tySet);

	p_tyC0007Notif ACCESS ADR(tyCommon.tyNotif);

	p_tyC0008MsgBox ACCESS ADR (tyP1024McSetAntiGap.tyMsgBoxHide);

	p_tyC0009Info ACCESS ADR(tyCommon.tyInfo);

	p_tyP1024McSetAntiGap ACCESS ADR(tyP1024McSetAntiGap.tyAntiGap);

	//Backup Param
	tyP1024McSetAntiGap.tyAntiGapBkUp	:= tyP1024McSetAntiGap.tyAntiGap;

END_ACTION
```

#### Act_OptP1024Navi.st
```iecst
ACTION Act_OptP1024Navi:

	tyP1024McSetAntiGap.tyNaviBack.tyBtnBack.bRtLk	:= tyCommon.tySet.tyBtnSave.bRtCompl;

	IF tyP1024McSetAntiGap.tyNaviBack.tyBtnBack.bRtCompl = TRUE THEN
		tyP1024McSetAntiGap.tyNaviBack.tyBtnBack.bRtCompl	:= FALSE;

		eChgPage	:= UIP1020McSetNavi;

	END_IF

END_ACTION
```
